ABB RAPID module: Module_Openhole.modx

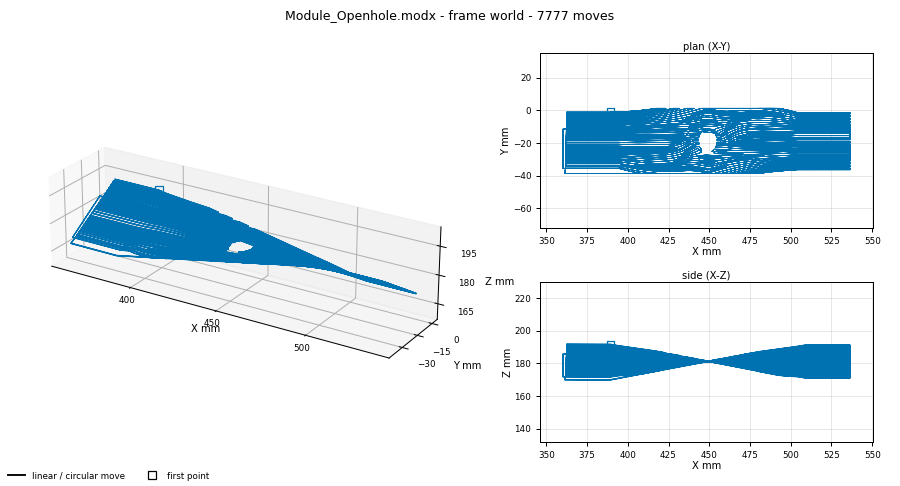
[picture p0: tool path of Module_Openhole.modx in frame world, 7777 of 7777 moves have a stored position in this frame; points joined in program order, loops and branches not executed]
MODULE Module_Openhole

	VAR robtarget Openhole_0 := [[389.38, -1.04, 191.45], [-0.232268, 0.667871, 0.694585, 0.132482], [0,0,0,0], [9E9, 9E9, 9E9, 9E9, 9E9, 9E9]];
	VAR robtarget Openhole_1 := [[394.38, -1.04, 190.58], [-0.220898, 0.671717, 0.697082, 0.118646], [0,0,0,0], [9E9, 9E9, 9E9, 9E9, 9E9, 9E9]];
	VAR robtarget Openhole_2 := [[406.26, -0.14, 188.9], [-0.1941, 0.679945, 0.702469, 0.080853], [0,0,0,0], [9E9, 9E9, 9E9, 9E9, 9E9, 9E9]];
	VAR robtarget Openhole_3 := [[415.11, 0.87, 187.62], [-0.173122, 0.685586, 0.705353, 0.049766], [0,0,0,0], [9E9, 9E9, 9E9, 9E9, 9E9, 9E9]];
	VAR robtarget Openhole_4 := [[417.07, 1.15, 187.33], [-0.16843, 0.686754, 0.705828, 0.042511], [0,0,0,0], [9E9, 9E9, 9E9, 9E9, 9E9, 9E9]];
	VAR robtarget Openhole_5 := [[417.57, 1.3, 187.28], [-0.167467, 0.68699, 0.70595, 0.040437], [0,0,0,0], [9E9, 9E9, 9E9, 9E9, 9E9, 9E9]];
	VAR robtarget Openhole_6 := [[423.41, 1.3, 186.14], [-0.150369, 0.690933, 0.706792, 0.021083], [0,0,0,0], [9E9, 9E9, 9E9, 9E9, 9E9, 9E9]];
	VAR robtarget Openhole_7 := [[422.92, 1.19, 186.21], [-0.151474, 0.690692, 0.70673, 0.023069], [0,0,0,0], [9E9, 9E9, 9E9, 9E9, 9E9, 9E9]];
	VAR robtarget Openhole_8 := [[416.08, 0.05, 187.17], [-0.167887, 0.686887, 0.705392, 0.04921], [0,0,0,0], [9E9, 9E9, 9E9, 9E9, 9E9, 9E9]];
	VAR robtarget Openhole_9 := [[407.72, -0.93, 188.32], [-0.187933, 0.681675, 0.702703, 0.078791], [0,0,0,0], [9E9, 9E9, 9E9, 9E9, 9E9, 9E9]];
	VAR robtarget Openhole_10 := [[395.86, -1.84, 189.92], [-0.215169, 0.673574, 0.697401, 0.116758], [0,0,0,0], [9E9, 9E9, 9E9, 9E9, 9E9, 9E9]];
	VAR robtarget Openhole_11 := [[394.37, -1.93, 190.11], [-0.218405, 0.672532, 0.696636, 0.121237], [0,0,0,0], [9E9, 9E9, 9E9, 9E9, 9E9, 9E9]];
	VAR robtarget Openhole_12 := [[389.38, -1.93, 190.93], [-0.229838, 0.668711, 0.694097, 0.135014], [0,0,0,0], [9E9, 9E9, 9E9, 9E9, 9E9, 9E9]];
	VAR robtarget Openhole_13 := [[362.38, -1.93, 191.02], [-0.183051, 0.683002, 0.683002, 0.183051], [0,0,0,0], [9E9, 9E9, 9E9, 9E9, 9E9, 9E9]];
	VAR robtarget Openhole_14 := [[362.37, -2.82, 190.51], [-0.183051, 0.683002, 0.683002, 0.183051], [0,0,0,0], [9E9, 9E9, 9E9, 9E9, 9E9, 9E9]];
	VAR robtarget Openhole_15 := [[374.37, -2.82, 190.47], [-0.183051, 0.683002, 0.683002, 0.183051], [0,0,0,0], [9E9, 9E9, 9E9, 9E9, 9E9, 9E9]];
	VAR robtarget Openhole_16 := [[389.37, -2.82, 190.42], [-0.227419, 0.669538, 0.693603, 0.137529], [0,0,0,0], [9E9, 9E9, 9E9, 9E9, 9E9, 9E9]];
	VAR robtarget Openhole_17 := [[394.37, -2.82, 189.64], [-0.215931, 0.67333, 0.696182, 0.12382], [0,0,0,0], [9E9, 9E9, 9E9, 9E9, 9E9, 9E9]];
	VAR robtarget Openhole_18 := [[408.22, -1.78, 187.89], [-0.184033, 0.682738, 0.702585, 0.079843], [0,0,0,0], [9E9, 9E9, 9E9, 9E9, 9E9, 9E9]];
	VAR robtarget Openhole_19 := [[416.11, -0.88, 186.87], [-0.164956, 0.687597, 0.705187, 0.052065], [0,0,0,0], [9E9, 9E9, 9E9, 9E9, 9E9, 9E9]];
	VAR robtarget Openhole_20 := [[422.95, 0.24, 185.96], [-0.148411, 0.691357, 0.706629, 0.025979], [0,0,0,0], [9E9, 9E9, 9E9, 9E9, 9E9, 9E9]];
	VAR robtarget Openhole_21 := [[427.32, 1.15, 185.34], [-0.138034, 0.693503, 0.707057, 0.008389], [0,0,0,0], [9E9, 9E9, 9E9, 9E9, 9E9, 9E9]];
	VAR robtarget Openhole_22 := [[427.8, 1.3, 185.28], [-0.137012, 0.693706, 0.707079, 0.006266], [0,0,0,0], [9E9, 9E9, 9E9, 9E9, 9E9, 9E9]];
	VAR robtarget Openhole_23 := [[431.7, 1.3, 184.52], [-0.124848, 0.695998, 0.707072, -0.007002], [0,0,0,0], [9E9, 9E9, 9E9, 9E9, 9E9, 9E9]];
	VAR robtarget Openhole_24 := [[431.22, 1.07, 184.57], [-0.125655, 0.695853, 0.707092, -0.004617], [0,0,0,0], [9E9, 9E9, 9E9, 9E9, 9E9, 9E9]];
	VAR robtarget Openhole_25 := [[423.96, -0.54, 185.58], [-0.142927, 0.692511, 0.706661, 0.025111], [0,0,0,0], [9E9, 9E9, 9E9, 9E9, 9E9, 9E9]];
	VAR robtarget Openhole_26 := [[417.11, -1.69, 186.44], [-0.159586, 0.688863, 0.70524, 0.051343], [0,0,0,0], [9E9, 9E9, 9E9, 9E9, 9E9, 9E9]];
	VAR robtarget Openhole_27 := [[409.22, -2.6, 187.41], [-0.178884, 0.684106, 0.702651, 0.079257], [0,0,0,0], [9E9, 9E9, 9E9, 9E9, 9E9, 9E9]];
	VAR robtarget Openhole_28 := [[394.87, -3.67, 189.12], [-0.212354, 0.674467, 0.695988, 0.124905], [0,0,0,0], [9E9, 9E9, 9E9, 9E9, 9E9, 9E9]];
	VAR robtarget Openhole_29 := [[394.36, -3.7, 189.17], [-0.21345, 0.674121, 0.695717, 0.126406], [0,0,0,0], [9E9, 9E9, 9E9, 9E9, 9E9, 9E9]];
	VAR robtarget Openhole_30 := [[389.37, -3.7, 189.91], [-0.224993, 0.670357, 0.693099, 0.140047], [0,0,0,0], [9E9, 9E9, 9E9, 9E9, 9E9, 9E9]];
	VAR robtarget Openhole_31 := [[362.37, -3.7, 190], [-0.183051, 0.683002, 0.683002, 0.183051], [0,0,0,0], [9E9, 9E9, 9E9, 9E9, 9E9, 9E9]];
	VAR robtarget Openhole_32 := [[362.37, -4.58, 189.49], [-0.183051, 0.683002, 0.683002, 0.183051], [0,0,0,0], [9E9, 9E9, 9E9, 9E9, 9E9, 9E9]];
	VAR robtarget Openhole_33 := [[374.37, -4.58, 189.45], [-0.183051, 0.683002, 0.683002, 0.183051], [0,0,0,0], [9E9, 9E9, 9E9, 9E9, 9E9, 9E9]];
	VAR robtarget Openhole_34 := [[389.37, -4.59, 189.4], [-0.222559, 0.671169, 0.692585, 0.142568], [0,0,0,0], [9E9, 9E9, 9E9, 9E9, 9E9, 9E9]];
	VAR robtarget Openhole_35 := [[394.36, -4.59, 188.71], [-0.210967, 0.674902, 0.69524, 0.129002], [0,0,0,0], [9E9, 9E9, 9E9, 9E9, 9E9, 9E9]];
	VAR robtarget Openhole_36 := [[409.73, -3.48, 186.99], [-0.17483, 0.685153, 0.702519, 0.080416], [0,0,0,0], [9E9, 9E9, 9E9, 9E9, 9E9, 9E9]];
	VAR robtarget Openhole_37 := [[417.63, -2.6, 186.08], [-0.155249, 0.689853, 0.70515, 0.052563], [0,0,0,0], [9E9, 9E9, 9E9, 9E9, 9E9, 9E9]];
	VAR robtarget Openhole_38 := [[424, -1.56, 185.32], [-0.13958, 0.693194, 0.706541, 0.028275], [0,0,0,0], [9E9, 9E9, 9E9, 9E9, 9E9, 9E9]];
	VAR robtarget Openhole_39 := [[430.79, -0.09, 184.44], [-0.12327, 0.696279, 0.707106, 0.000635], [0,0,0,0], [9E9, 9E9, 9E9, 9E9, 9E9, 9E9]];
	VAR robtarget Openhole_40 := [[435.6, 1.08, 183.72], [-0.111729, 0.698224, 0.706834, -0.019623], [0,0,0,0], [9E9, 9E9, 9E9, 9E9, 9E9, 9E9]];
	VAR robtarget Openhole_41 := [[436.08, 1.3, 183.66], [-0.110872, 0.698361, 0.706765, -0.021984], [0,0,0,0], [9E9, 9E9, 9E9, 9E9, 9E9, 9E9]];
	VAR robtarget Openhole_42 := [[440.9, 1.3, 182.71], [-0.095117, 0.70068, 0.706055, -0.038547], [0,0,0,0], [9E9, 9E9, 9E9, 9E9, 9E9, 9E9]];
	VAR robtarget Openhole_43 := [[440.43, 1.14, 182.79], [-0.096181, 0.700535, 0.706169, -0.036397], [0,0,0,0], [9E9, 9E9, 9E9, 9E9, 9E9, 9E9]];
	VAR robtarget Openhole_44 := [[431.79, -1.04, 184.1], [-0.11708, 0.697347, 0.707107, 0.000291], [0,0,0,0], [9E9, 9E9, 9E9, 9E9, 9E9, 9E9]];
	VAR robtarget Openhole_45 := [[425, -2.5, 184.94], [-0.133577, 0.694375, 0.706553, 0.027979], [0,0,0,0], [9E9, 9E9, 9E9, 9E9, 9E9, 9E9]];
	VAR robtarget Openhole_46 := [[418.62, -3.5, 185.66], [-0.149564, 0.691108, 0.705175, 0.052228], [0,0,0,0], [9E9, 9E9, 9E9, 9E9, 9E9, 9E9]];
	VAR robtarget Openhole_47 := [[410.22, -4.4, 186.57], [-0.170741, 0.686183, 0.702365, 0.081753], [0,0,0,0], [9E9, 9E9, 9E9, 9E9, 9E9, 9E9]];
	VAR robtarget Openhole_48 := [[394.37, -5.47, 188.24], [-0.208439, 0.675687, 0.694762, 0.131552], [0,0,0,0], [9E9, 9E9, 9E9, 9E9, 9E9, 9E9]];
	VAR robtarget Openhole_49 := [[389.37, -5.47, 188.89], [-0.220121, 0.671972, 0.692061, 0.14509], [0,0,0,0], [9E9, 9E9, 9E9, 9E9, 9E9, 9E9]];
	VAR robtarget Openhole_50 := [[362.37, -5.47, 188.98], [-0.183051, 0.683002, 0.683002, 0.183051], [0,0,0,0], [9E9, 9E9, 9E9, 9E9, 9E9, 9E9]];
	VAR robtarget Openhole_51 := [[362.37, -6.37, 188.45], [-0.183051, 0.683002, 0.683002, 0.183051], [0,0,0,0], [9E9, 9E9, 9E9, 9E9, 9E9, 9E9]];
	VAR robtarget Openhole_52 := [[374.37, -6.37, 188.42], [-0.183051, 0.683002, 0.683002, 0.183051], [0,0,0,0], [9E9, 9E9, 9E9, 9E9, 9E9, 9E9]];
	VAR robtarget Openhole_53 := [[389.37, -6.37, 188.37], [-0.217615, 0.672788, 0.691514, 0.147675], [0,0,0,0], [9E9, 9E9, 9E9, 9E9, 9E9, 9E9]];
	VAR robtarget Openhole_54 := [[394.35, -6.37, 187.76], [-0.205904, 0.676464, 0.694247, 0.134242], [0,0,0,0], [9E9, 9E9, 9E9, 9E9, 9E9, 9E9]];
	VAR robtarget Openhole_55 := [[411.74, -5.23, 186.06], [-0.163934, 0.687841, 0.702611, 0.079612], [0,0,0,0], [9E9, 9E9, 9E9, 9E9, 9E9, 9E9]];
	VAR robtarget Openhole_56 := [[420.15, -4.36, 185.18], [-0.142311, 0.692638, 0.705338, 0.049989], [0,0,0,0], [9E9, 9E9, 9E9, 9E9, 9E9, 9E9]];
	VAR robtarget Openhole_57 := [[427.03, -3.3, 184.44], [-0.12476, 0.696014, 0.706707, 0.023772], [0,0,0,0], [9E9, 9E9, 9E9, 9E9, 9E9, 9E9]];
	VAR robtarget Openhole_58 := [[432.87, -2.08, 183.75], [-0.110304, 0.69845, 0.707107, 0.000048], [0,0,0,0], [9E9, 9E9, 9E9, 9E9, 9E9, 9E9]];
	VAR robtarget Openhole_59 := [[441.01, 0.05, 182.59], [-0.090709, 0.701264, 0.706248, -0.034832], [0,0,0,0], [9E9, 9E9, 9E9, 9E9, 9E9, 9E9]];
	VAR robtarget Openhole_60 := [[444.81, 1.13, 181.94], [-0.081605, 0.702382, 0.705237, -0.051387], [0,0,0,0], [9E9, 9E9, 9E9, 9E9, 9E9, 9E9]];
	VAR robtarget Openhole_61 := [[445.28, 1.3, 181.86], [-0.080561, 0.702503, 0.705076, -0.053548], [0,0,0,0], [9E9, 9E9, 9E9, 9E9, 9E9, 9E9]];
	VAR robtarget Openhole_62 := [[492.93, 1.3, 172.53], [0.078494, 0.702737, 0.678213, -0.200067], [0,0,0,0], [9E9, 9E9, 9E9, 9E9, 9E9, 9E9]];
	VAR robtarget Openhole_63 := [[497.81, 0.35, 172.02], [0.095716, 0.700599, 0.675215, -0.209963], [0,0,0,0], [9E9, 9E9, 9E9, 9E9, 9E9, 9E9]];
	VAR robtarget Openhole_64 := [[502.17, -0.75, 171.76], [0.111656, 0.698236, 0.672857, -0.217402], [0,0,0,0], [9E9, 9E9, 9E9, 9E9, 9E9, 9E9]];
	VAR robtarget Openhole_65 := [[503.61, -1.18, 171.73], [0.117001, 0.69736, 0.672147, -0.219587], [0,0,0,0], [9E9, 9E9, 9E9, 9E9, 9E9, 9E9]];
	VAR robtarget Openhole_66 := [[504.32, -1.34, 171.7], [0.119471, 0.696941, 0.67175, -0.220799], [0,0,0,0], [9E9, 9E9, 9E9, 9E9, 9E9, 9E9]];
	VAR robtarget Openhole_67 := [[509.31, -1.34, 170.85], [0.183051, 0.683002, 0.683002, -0.183051], [0,0,0,0], [9E9, 9E9, 9E9, 9E9, 9E9, 9E9]];
	VAR robtarget Openhole_68 := [[536.31, -1.34, 170.76], [0.183051, 0.683002, 0.683002, -0.183051], [0,0,0,0], [9E9, 9E9, 9E9, 9E9, 9E9, 9E9]];
	VAR robtarget Openhole_69 := [[536.31, -1.86, 171.07], [0.183051, 0.683002, 0.683002, -0.183051], [0,0,0,0], [9E9, 9E9, 9E9, 9E9, 9E9, 9E9]];
	VAR robtarget Openhole_70 := [[509.31, -1.86, 171.15], [0.183051, 0.683002, 0.683002, -0.183051], [0,0,0,0], [9E9, 9E9, 9E9, 9E9, 9E9, 9E9]];
	VAR robtarget Openhole_71 := [[504.32, -1.86, 171.98], [0.120994, 0.696678, 0.672232, -0.219328], [0,0,0,0], [9E9, 9E9, 9E9, 9E9, 9E9, 9E9]];
	VAR robtarget Openhole_72 := [[503.45, -1.68, 172.02], [0.118004, 0.697191, 0.672724, -0.217813], [0,0,0,0], [9E9, 9E9, 9E9, 9E9, 9E9, 9E9]];
	VAR robtarget Openhole_73 := [[502.98, -1.51, 172.02], [0.116192, 0.697495, 0.672938, -0.217151], [0,0,0,0], [9E9, 9E9, 9E9, 9E9, 9E9, 9E9]];
	VAR robtarget Openhole_74 := [[498.64, -0.34, 172.19], [0.100205, 0.699971, 0.675206, -0.209992], [0,0,0,0], [9E9, 9E9, 9E9, 9E9, 9E9, 9E9]];
	VAR robtarget Openhole_75 := [[493.76, 0.68, 172.63], [0.082548, 0.702272, 0.678031, -0.200682], [0,0,0,0], [9E9, 9E9, 9E9, 9E9, 9E9, 9E9]];
	VAR robtarget Openhole_76 := [[490.83, 1.18, 172.99], [0.071986, 0.703433, 0.679827, -0.194513], [0,0,0,0], [9E9, 9E9, 9E9, 9E9, 9E9, 9E9]];
	VAR robtarget Openhole_77 := [[490.33, 1.3, 173.04], [0.070413, 0.703592, 0.680176, -0.193289], [0,0,0,0], [9E9, 9E9, 9E9, 9E9, 9E9, 9E9]];
	VAR robtarget Openhole_78 := [[480.37, 1.3, 174.99], [0.038399, 0.706063, 0.687393, -0.165806], [0,0,0,0], [9E9, 9E9, 9E9, 9E9, 9E9, 9E9]];
	VAR robtarget Openhole_79 := [[486.26, 0.75, 174.03], [0.058914, 0.704648, 0.683556, -0.180974], [0,0,0,0], [9E9, 9E9, 9E9, 9E9, 9E9, 9E9]];
	VAR robtarget Openhole_80 := [[492.15, -0.08, 173.25], [0.079897, 0.702578, 0.679886, -0.194305], [0,0,0,0], [9E9, 9E9, 9E9, 9E9, 9E9, 9E9]];
	VAR robtarget Openhole_81 := [[497.53, -1.09, 172.74], [0.099178, 0.700117, 0.676708, -0.2051], [0,0,0,0], [9E9, 9E9, 9E9, 9E9, 9E9, 9E9]];
	VAR robtarget Openhole_82 := [[502.86, -2.42, 172.5], [0.118516, 0.697104, 0.673843, -0.214326], [0,0,0,0], [9E9, 9E9, 9E9, 9E9, 9E9, 9E9]];
	VAR robtarget Openhole_83 := [[503.83, -2.67, 172.48], [0.121975, 0.696507, 0.673336, -0.215915], [0,0,0,0], [9E9, 9E9, 9E9, 9E9, 9E9, 9E9]];
	VAR robtarget Openhole_84 := [[504.4, -2.79, 172.45], [0.123921, 0.696164, 0.673011, -0.216923], [0,0,0,0], [9E9, 9E9, 9E9, 9E9, 9E9, 9E9]];
	VAR robtarget Openhole_85 := [[509.32, -2.79, 171.69], [0.183051, 0.683002, 0.683002, -0.183051], [0,0,0,0], [9E9, 9E9, 9E9, 9E9, 9E9, 9E9]];
	VAR robtarget Openhole_86 := [[536.32, -2.79, 171.6], [0.183051, 0.683002, 0.683002, -0.183051], [0,0,0,0], [9E9, 9E9, 9E9, 9E9, 9E9, 9E9]];
	VAR robtarget Openhole_87 := [[536.32, -3.66, 172.1], [0.183051, 0.683002, 0.683002, -0.183051], [0,0,0,0], [9E9, 9E9, 9E9, 9E9, 9E9, 9E9]];
	VAR robtarget Openhole_88 := [[509.32, -3.66, 172.19], [0.183051, 0.683002, 0.683002, -0.183051], [0,0,0,0], [9E9, 9E9, 9E9, 9E9, 9E9, 9E9]];
	VAR robtarget Openhole_89 := [[504.32, -3.66, 172.93], [0.126217, 0.695751, 0.67386, -0.214271], [0,0,0,0], [9E9, 9E9, 9E9, 9E9, 9E9, 9E9]];
	VAR robtarget Openhole_90 := [[503.61, -3.55, 172.97], [0.123897, 0.696168, 0.67429, -0.212914], [0,0,0,0], [9E9, 9E9, 9E9, 9E9, 9E9, 9E9]];
	VAR robtarget Openhole_91 := [[496.78, -2.08, 173.32], [0.099881, 0.700017, 0.678136, -0.200327], [0,0,0,0], [9E9, 9E9, 9E9, 9E9, 9E9, 9E9]];
	VAR robtarget Openhole_92 := [[490.88, -1.1, 173.89], [0.079095, 0.702669, 0.681676, -0.187931], [0,0,0,0], [9E9, 9E9, 9E9, 9E9, 9E9, 9E9]];
	VAR robtarget Openhole_93 := [[484.49, -0.34, 174.74], [0.056636, 0.704835, 0.685689, -0.172716], [0,0,0,0], [9E9, 9E9, 9E9, 9E9, 9E9, 9E9]];
	VAR robtarget Openhole_94 := [[478.08, 0.04, 175.78], [0.034605, 0.70626, 0.6898, -0.155485], [0,0,0,0], [9E9, 9E9, 9E9, 9E9, 9E9, 9E9]];
	VAR robtarget Openhole_95 := [[475.62, 0.08, 176.23], [0.026334, 0.706616, 0.691382, -0.148292], [0,0,0,0], [9E9, 9E9, 9E9, 9E9, 9E9, 9E9]];
	VAR robtarget Openhole_96 := [[475.13, 0.08, 176.32], [0.024701, 0.706675, 0.691699, -0.14681], [0,0,0,0], [9E9, 9E9, 9E9, 9E9, 9E9, 9E9]];
	VAR robtarget Openhole_97 := [[468.75, -0.12, 177.53], [0.003925, 0.707096, 0.695696, -0.126519], [0,0,0,0], [9E9, 9E9, 9E9, 9E9, 9E9, 9E9]];
	VAR robtarget Openhole_98 := [[461.39, -0.49, 178.91], [-0.019926, 0.706826, 0.699751, -0.101727], [0,0,0,0], [9E9, 9E9, 9E9, 9E9, 9E9, 9E9]];
	VAR robtarget Openhole_99 := [[460.9, -0.5, 179], [-0.021584, 0.706777, 0.699986, -0.100097], [0,0,0,0], [9E9, 9E9, 9E9, 9E9, 9E9, 9E9]];
	VAR robtarget Openhole_100 := [[459.91, -0.49, 179.18], [-0.024971, 0.706666, 0.700437, -0.096889], [0,0,0,0], [9E9, 9E9, 9E9, 9E9, 9E9, 9E9]];
	VAR robtarget Openhole_101 := [[457.94, -0.41, 179.52], [-0.031979, 0.706383, 0.701269, -0.090672], [0,0,0,0], [9E9, 9E9, 9E9, 9E9, 9E9, 9E9]];
	VAR robtarget Openhole_102 := [[456.96, -0.33, 179.69], [-0.035593, 0.70621, 0.701651, -0.087669], [0,0,0,0], [9E9, 9E9, 9E9, 9E9, 9E9, 9E9]];
	VAR robtarget Openhole_103 := [[455.49, -0.16, 179.94], [-0.041157, 0.705908, 0.702181, -0.083319], [0,0,0,0], [9E9, 9E9, 9E9, 9E9, 9E9, 9E9]];
	VAR robtarget Openhole_104 := [[454.52, -0.01, 180.11], [-0.044983, 0.705675, 0.702502, -0.080563], [0,0,0,0], [9E9, 9E9, 9E9, 9E9, 9E9, 9E9]];
	VAR robtarget Openhole_105 := [[453.55, 0.19, 180.28], [-0.048932, 0.705412, 0.702794, -0.077981], [0,0,0,0], [9E9, 9E9, 9E9, 9E9, 9E9, 9E9]];
	VAR robtarget Openhole_106 := [[453.08, 0.32, 180.37], [-0.050991, 0.705266, 0.702921, -0.076829], [0,0,0,0], [9E9, 9E9, 9E9, 9E9, 9E9, 9E9]];
	VAR robtarget Openhole_107 := [[451.65, 0.69, 180.62], [-0.057053, 0.704801, 0.703309, -0.07319], [0,0,0,0], [9E9, 9E9, 9E9, 9E9, 9E9, 9E9]];
	VAR robtarget Openhole_108 := [[451.16, 0.77, 180.71], [-0.058985, 0.704642, 0.703448, -0.071844], [0,0,0,0], [9E9, 9E9, 9E9, 9E9, 9E9, 9E9]];
	VAR robtarget Openhole_109 := [[450.68, 0.85, 180.81], [-0.060871, 0.704482, 0.70359, -0.070433], [0,0,0,0], [9E9, 9E9, 9E9, 9E9, 9E9, 9E9]];
	VAR robtarget Openhole_110 := [[450.19, 0.88, 180.9], [-0.062639, 0.704327, 0.703744, -0.06888], [0,0,0,0], [9E9, 9E9, 9E9, 9E9, 9E9, 9E9]];
	VAR robtarget Openhole_111 := [[449.7, 0.9, 180.99], [-0.06438, 0.70417, 0.703897, -0.067293], [0,0,0,0], [9E9, 9E9, 9E9, 9E9, 9E9, 9E9]];
	VAR robtarget Openhole_112 := [[449.21, 0.87, 181.09], [-0.065931, 0.704026, 0.704065, -0.065521], [0,0,0,0], [9E9, 9E9, 9E9, 9E9, 9E9, 9E9]];
	VAR robtarget Openhole_113 := [[448.72, 0.81, 181.18], [-0.067402, 0.703887, 0.704233, -0.063683], [0,0,0,0], [9E9, 9E9, 9E9, 9E9, 9E9, 9E9]];
	VAR robtarget Openhole_114 := [[447.76, 0.61, 181.36], [-0.069985, 0.703635, 0.704579, -0.05974], [0,0,0,0], [9E9, 9E9, 9E9, 9E9, 9E9, 9E9]];
	VAR robtarget Openhole_115 := [[446.8, 0.36, 181.54], [-0.072379, 0.703393, 0.704912, -0.055673], [0,0,0,0], [9E9, 9E9, 9E9, 9E9, 9E9, 9E9]];
	VAR robtarget Openhole_116 := [[438.73, -1.98, 182.8], [-0.091604, 0.701148, 0.706814, -0.02033], [0,0,0,0], [9E9, 9E9, 9E9, 9E9, 9E9, 9E9]];
	VAR robtarget Openhole_117 := [[433.43, -3.29, 183.47], [-0.104537, 0.699337, 0.707104, 0.002109], [0,0,0,0], [9E9, 9E9, 9E9, 9E9, 9E9, 9E9]];
	VAR robtarget Openhole_118 := [[427.08, -4.48, 184.18], [-0.120798, 0.696712, 0.706573, 0.027462], [0,0,0,0], [9E9, 9E9, 9E9, 9E9, 9E9, 9E9]];
	VAR robtarget Openhole_119 := [[419.69, -5.48, 184.93], [-0.140178, 0.693073, 0.704958, 0.055089], [0,0,0,0], [9E9, 9E9, 9E9, 9E9, 9E9, 9E9]];
	VAR robtarget Openhole_120 := [[409.77, -6.33, 185.9], [-0.166065, 0.68733, 0.701464, 0.089152], [0,0,0,0], [9E9, 9E9, 9E9, 9E9, 9E9, 9E9]];
	VAR robtarget Openhole_121 := [[394.35, -7.26, 187.29], [-0.203395, 0.677223, 0.69374, 0.136838], [0,0,0,0], [9E9, 9E9, 9E9, 9E9, 9E9, 9E9]];
	VAR robtarget Openhole_122 := [[389.37, -7.26, 187.86], [-0.215162, 0.673577, 0.69097, 0.150202], [0,0,0,0], [9E9, 9E9, 9E9, 9E9, 9E9, 9E9]];
	VAR robtarget Openhole_123 := [[362.37, -7.26, 187.94], [-0.183051, 0.683002, 0.683002, 0.183051], [0,0,0,0], [9E9, 9E9, 9E9, 9E9, 9E9, 9E9]];
	VAR robtarget Openhole_124 := [[362.37, -8.14, 187.43], [-0.183051, 0.683002, 0.683002, 0.183051], [0,0,0,0], [9E9, 9E9, 9E9, 9E9, 9E9, 9E9]];
	VAR robtarget Openhole_125 := [[374.36, -8.14, 187.4], [-0.183051, 0.683002, 0.683002, 0.183051], [0,0,0,0], [9E9, 9E9, 9E9, 9E9, 9E9, 9E9]];
	VAR robtarget Openhole_126 := [[389.36, -8.14, 187.35], [-0.212703, 0.674357, 0.690416, 0.152729], [0,0,0,0], [9E9, 9E9, 9E9, 9E9, 9E9, 9E9]];
	VAR robtarget Openhole_127 := [[394.35, -8.14, 186.83], [-0.200864, 0.677978, 0.693227, 0.139415], [0,0,0,0], [9E9, 9E9, 9E9, 9E9, 9E9, 9E9]];
	VAR robtarget Openhole_128 := [[411.28, -7.19, 185.4], [-0.159238, 0.688944, 0.701709, 0.087206], [0,0,0,0], [9E9, 9E9, 9E9, 9E9, 9E9, 9E9]];
	VAR robtarget Openhole_129 := [[421.2, -6.39, 184.49], [-0.132741, 0.694536, 0.705109, 0.053119], [0,0,0,0], [9E9, 9E9, 9E9, 9E9, 9E9, 9E9]];
	VAR robtarget Openhole_130 := [[429.59, -5.33, 183.67], [-0.110165, 0.698472, 0.70677, 0.021825], [0,0,0,0], [9E9, 9E9, 9E9, 9E9, 9E9, 9E9]];
	VAR robtarget Openhole_131 := [[435.95, -4.17, 182.98], [-0.09353, 0.700894, 0.707098, -0.003575], [0,0,0,0], [9E9, 9E9, 9E9, 9E9, 9E9, 9E9]];
	VAR robtarget Openhole_132 := [[441.25, -2.83, 182.32], [-0.08048, 0.702512, 0.706625, -0.026102], [0,0,0,0], [9E9, 9E9, 9E9, 9E9, 9E9, 9E9]];
	VAR robtarget Openhole_133 := [[446.48, -1.34, 181.55], [-0.06789, 0.70384, 0.705409, -0.048969], [0,0,0,0], [9E9, 9E9, 9E9, 9E9, 9E9, 9E9]];
	VAR robtarget Openhole_134 := [[447.44, -1.11, 181.39], [-0.065397, 0.704076, 0.705118, -0.052996], [0,0,0,0], [9E9, 9E9, 9E9, 9E9, 9E9, 9E9]];
	VAR robtarget Openhole_135 := [[447.92, -1.01, 181.31], [-0.064108, 0.704195, 0.704966, -0.054981], [0,0,0,0], [9E9, 9E9, 9E9, 9E9, 9E9, 9E9]];
	VAR robtarget Openhole_136 := [[448.41, -0.92, 181.22], [-0.062761, 0.704316, 0.704812, -0.056924], [0,0,0,0], [9E9, 9E9, 9E9, 9E9, 9E9, 9E9]];
	VAR robtarget Openhole_137 := [[448.9, -0.86, 181.14], [-0.061324, 0.704443, 0.704658, -0.058803], [0,0,0,0], [9E9, 9E9, 9E9, 9E9, 9E9, 9E9]];
	VAR robtarget Openhole_138 := [[449.39, -0.83, 181.05], [-0.059734, 0.704579, 0.70451, -0.060549], [0,0,0,0], [9E9, 9E9, 9E9, 9E9, 9E9, 9E9]];
	VAR robtarget Openhole_139 := [[449.88, -0.83, 180.97], [-0.058081, 0.704717, 0.704362, -0.06224], [0,0,0,0], [9E9, 9E9, 9E9, 9E9, 9E9, 9E9]];
	VAR robtarget Openhole_140 := [[450.37, -0.87, 180.88], [-0.056288, 0.704863, 0.704224, -0.063781], [0,0,0,0], [9E9, 9E9, 9E9, 9E9, 9E9, 9E9]];
	VAR robtarget Openhole_141 := [[450.86, -0.92, 180.8], [-0.054451, 0.705007, 0.704088, -0.065265], [0,0,0,0], [9E9, 9E9, 9E9, 9E9, 9E9, 9E9]];
	VAR robtarget Openhole_142 := [[451.35, -1, 180.71], [-0.052532, 0.705153, 0.703959, -0.066646], [0,0,0,0], [9E9, 9E9, 9E9, 9E9, 9E9, 9E9]];
	VAR robtarget Openhole_143 := [[452.32, -1.2, 180.55], [-0.048584, 0.705436, 0.703708, -0.069247], [0,0,0,0], [9E9, 9E9, 9E9, 9E9, 9E9, 9E9]];
	VAR robtarget Openhole_144 := [[452.8, -1.31, 180.47], [-0.046578, 0.705571, 0.703584, -0.070498], [0,0,0,0], [9E9, 9E9, 9E9, 9E9, 9E9, 9E9]];
	VAR robtarget Openhole_145 := [[455.22, -1.78, 180.09], [-0.036759, 0.706151, 0.702891, -0.077096], [0,0,0,0], [9E9, 9E9, 9E9, 9E9, 9E9, 9E9]];
	VAR robtarget Openhole_146 := [[459.15, -2.25, 179.48], [-0.021814, 0.70677, 0.701532, -0.088615], [0,0,0,0], [9E9, 9E9, 9E9, 9E9, 9E9, 9E9]];
	VAR robtarget Openhole_147 := [[459.64, -2.28, 179.4], [-0.020033, 0.706823, 0.701337, -0.090147], [0,0,0,0], [9E9, 9E9, 9E9, 9E9, 9E9, 9E9]];
	VAR robtarget Openhole_148 := [[460.13, -2.3, 179.32], [-0.018281, 0.70687, 0.701135, -0.091707], [0,0,0,0], [9E9, 9E9, 9E9, 9E9, 9E9, 9E9]];
	VAR robtarget Openhole_149 := [[461.12, -2.32, 179.17], [-0.014848, 0.706951, 0.700711, -0.094889], [0,0,0,0], [9E9, 9E9, 9E9, 9E9, 9E9, 9E9]];
	VAR robtarget Openhole_150 := [[466.05, -2.11, 178.34], [0.001206, 0.707106, 0.698251, -0.111559], [0,0,0,0], [9E9, 9E9, 9E9, 9E9, 9E9, 9E9]];
	VAR robtarget Openhole_151 := [[473.41, -1.61, 177.02], [0.024393, 0.706686, 0.693856, -0.136249], [0,0,0,0], [9E9, 9E9, 9E9, 9E9, 9E9, 9E9]];
	VAR robtarget Openhole_152 := [[476.86, -1.55, 176.43], [0.035645, 0.706208, 0.691685, -0.146871], [0,0,0,0], [9E9, 9E9, 9E9, 9E9, 9E9, 9E9]];
	VAR robtarget Openhole_153 := [[477.35, -1.55, 176.35], [0.037279, 0.706123, 0.691373, -0.148336], [0,0,0,0], [9E9, 9E9, 9E9, 9E9, 9E9, 9E9]];
	VAR robtarget Openhole_154 := [[483.28, -1.79, 175.43], [0.057281, 0.704783, 0.687617, -0.164874], [0,0,0,0], [9E9, 9E9, 9E9, 9E9, 9E9, 9E9]];
	VAR robtarget Openhole_155 := [[489.2, -2.35, 174.66], [0.077729, 0.702822, 0.683906, -0.179645], [0,0,0,0], [9E9, 9E9, 9E9, 9E9, 9E9, 9E9]];
	VAR robtarget Openhole_156 := [[496.1, -3.34, 174], [0.101648, 0.699763, 0.67971, -0.194921], [0,0,0,0], [9E9, 9E9, 9E9, 9E9, 9E9, 9E9]];
	VAR robtarget Openhole_157 := [[501.51, -4.28, 173.65], [0.120102, 0.696833, 0.67651, -0.205751], [0,0,0,0], [9E9, 9E9, 9E9, 9E9, 9E9, 9E9]];
	VAR robtarget Openhole_158 := [[503.48, -4.58, 173.53], [0.126548, 0.695691, 0.675311, -0.209654], [0,0,0,0], [9E9, 9E9, 9E9, 9E9, 9E9, 9E9]];
	VAR robtarget Openhole_159 := [[504.32, -4.67, 173.46], [0.129153, 0.695212, 0.674761, -0.211419], [0,0,0,0], [9E9, 9E9, 9E9, 9E9, 9E9, 9E9]];
	VAR robtarget Openhole_160 := [[509.32, -4.67, 172.77], [0.183051, 0.683002, 0.683002, -0.183051], [0,0,0,0], [9E9, 9E9, 9E9, 9E9, 9E9, 9E9]];
	VAR robtarget Openhole_161 := [[536.32, -4.67, 172.69], [0.183051, 0.683002, 0.683002, -0.183051], [0,0,0,0], [9E9, 9E9, 9E9, 9E9, 9E9, 9E9]];
	VAR robtarget Openhole_162 := [[536.32, -5.62, 173.24], [0.183051, 0.683002, 0.683002, -0.183051], [0,0,0,0], [9E9, 9E9, 9E9, 9E9, 9E9, 9E9]];
	VAR robtarget Openhole_163 := [[524.32, -5.62, 173.27], [0.183051, 0.683002, 0.683002, -0.183051], [0,0,0,0], [9E9, 9E9, 9E9, 9E9, 9E9, 9E9]];
	VAR robtarget Openhole_164 := [[509.32, -5.62, 173.32], [0.183051, 0.683002, 0.683002, -0.183051], [0,0,0,0], [9E9, 9E9, 9E9, 9E9, 9E9, 9E9]];
	VAR robtarget Openhole_165 := [[504.32, -5.62, 173.97], [0.1319, 0.694696, 0.675605, -0.208705], [0,0,0,0], [9E9, 9E9, 9E9, 9E9, 9E9, 9E9]];
	VAR robtarget Openhole_166 := [[503.82, -5.61, 174.03], [0.130493, 0.694962, 0.675962, -0.207547], [0,0,0,0], [9E9, 9E9, 9E9, 9E9, 9E9, 9E9]];
	VAR robtarget Openhole_167 := [[498.86, -5.11, 174.43], [0.115013, 0.69769, 0.679175, -0.196776], [0,0,0,0], [9E9, 9E9, 9E9, 9E9, 9E9, 9E9]];
	VAR robtarget Openhole_168 := [[489.97, -3.94, 175.16], [0.084986, 0.701981, 0.684607, -0.176954], [0,0,0,0], [9E9, 9E9, 9E9, 9E9, 9E9, 9E9]];
	VAR robtarget Openhole_169 := [[483.54, -3.35, 175.9], [0.063031, 0.704292, 0.68858, -0.160802], [0,0,0,0], [9E9, 9E9, 9E9, 9E9, 9E9, 9E9]];
	VAR robtarget Openhole_170 := [[478.1, -3.15, 176.67], [0.044814, 0.705685, 0.691968, -0.145535], [0,0,0,0], [9E9, 9E9, 9E9, 9E9, 9E9, 9E9]];
	VAR robtarget Openhole_171 := [[477.6, -3.15, 176.74], [0.043193, 0.705786, 0.692276, -0.144062], [0,0,0,0], [9E9, 9E9, 9E9, 9E9, 9E9, 9E9]];
	VAR robtarget Openhole_172 := [[477.11, -3.15, 176.82], [0.041573, 0.705884, 0.692583, -0.142581], [0,0,0,0], [9E9, 9E9, 9E9, 9E9, 9E9, 9E9]];
	VAR robtarget Openhole_173 := [[471.68, -3.36, 177.69], [0.024304, 0.706689, 0.695916, -0.125306], [0,0,0,0], [9E9, 9E9, 9E9, 9E9, 9E9, 9E9]];
	VAR robtarget Openhole_174 := [[462.34, -4.17, 179.2], [-0.004601, 0.707092, 0.700988, -0.092824], [0,0,0,0], [9E9, 9E9, 9E9, 9E9, 9E9, 9E9]];
	VAR robtarget Openhole_175 := [[459.87, -4.23, 179.56], [-0.012811, 0.706991, 0.702042, -0.084482], [0,0,0,0], [9E9, 9E9, 9E9, 9E9, 9E9, 9E9]];
	VAR robtarget Openhole_176 := [[459.37, -4.22, 179.63], [-0.014523, 0.706958, 0.702234, -0.082867], [0,0,0,0], [9E9, 9E9, 9E9, 9E9, 9E9, 9E9]];
	VAR robtarget Openhole_177 := [[458.38, -4.18, 179.77], [-0.018029, 0.706877, 0.702599, -0.079714], [0,0,0,0], [9E9, 9E9, 9E9, 9E9, 9E9, 9E9]];
	VAR robtarget Openhole_178 := [[457.39, -4.11, 179.91], [-0.021647, 0.706775, 0.702938, -0.076673], [0,0,0,0], [9E9, 9E9, 9E9, 9E9, 9E9, 9E9]];
	VAR robtarget Openhole_179 := [[452.98, -3.48, 180.52], [-0.038778, 0.706043, 0.704209, -0.06395], [0,0,0,0], [9E9, 9E9, 9E9, 9E9, 9E9, 9E9]];
	VAR robtarget Openhole_180 := [[451.03, -3.16, 180.8], [-0.046477, 0.705578, 0.704691, -0.058395], [0,0,0,0], [9E9, 9E9, 9E9, 9E9, 9E9, 9E9]];
	VAR robtarget Openhole_181 := [[450.54, -3.1, 180.88], [-0.048352, 0.705452, 0.70481, -0.056941], [0,0,0,0], [9E9, 9E9, 9E9, 9E9, 9E9, 9E9]];
	VAR robtarget Openhole_182 := [[449.55, -3.01, 181.03], [-0.051994, 0.705193, 0.705049, -0.0539], [0,0,0,0], [9E9, 9E9, 9E9, 9E9, 9E9, 9E9]];
	VAR robtarget Openhole_183 := [[449.06, -3, 181.11], [-0.053711, 0.705064, 0.705173, -0.052264], [0,0,0,0], [9E9, 9E9, 9E9, 9E9, 9E9, 9E9]];
	VAR robtarget Openhole_184 := [[448.57, -3, 181.18], [-0.055374, 0.704935, 0.705296, -0.050571], [0,0,0,0], [9E9, 9E9, 9E9, 9E9, 9E9, 9E9]];
	VAR robtarget Openhole_185 := [[448.07, -3.04, 181.26], [-0.056913, 0.704813, 0.705423, -0.048764], [0,0,0,0], [9E9, 9E9, 9E9, 9E9, 9E9, 9E9]];
	VAR robtarget Openhole_186 := [[447.58, -3.09, 181.33], [-0.05842, 0.704689, 0.705548, -0.04693], [0,0,0,0], [9E9, 9E9, 9E9, 9E9, 9E9, 9E9]];
	VAR robtarget Openhole_187 := [[447.09, -3.15, 181.41], [-0.05986, 0.704568, 0.705671, -0.045042], [0,0,0,0], [9E9, 9E9, 9E9, 9E9, 9E9, 9E9]];
	VAR robtarget Openhole_188 := [[446.11, -3.31, 181.55], [-0.062631, 0.704328, 0.705907, -0.041182], [0,0,0,0], [9E9, 9E9, 9E9, 9E9, 9E9, 9E9]];
	VAR robtarget Openhole_189 := [[437.9, -5.24, 182.58], [-0.083589, 0.702149, 0.707076, -0.006649], [0,0,0,0], [9E9, 9E9, 9E9, 9E9, 9E9, 9E9]];
	VAR robtarget Openhole_190 := [[431.53, -6.32, 183.24], [-0.100765, 0.69989, 0.706862, 0.018588], [0,0,0,0], [9E9, 9E9, 9E9, 9E9, 9E9, 9E9]];
	VAR robtarget Openhole_191 := [[423.12, -7.3, 184.02], [-0.123999, 0.69615, 0.705352, 0.049786], [0,0,0,0], [9E9, 9E9, 9E9, 9E9, 9E9, 9E9]];
	VAR robtarget Openhole_192 := [[413.19, -8.06, 184.88], [-0.151113, 0.690771, 0.702098, 0.084016], [0,0,0,0], [9E9, 9E9, 9E9, 9E9, 9E9, 9E9]];
	VAR robtarget Openhole_193 := [[394.36, -9.02, 186.36], [-0.198303, 0.678731, 0.692709, 0.141966], [0,0,0,0], [9E9, 9E9, 9E9, 9E9, 9E9, 9E9]];
	VAR robtarget Openhole_194 := [[389.36, -9.02, 186.84], [-0.210239, 0.675129, 0.689852, 0.155257], [0,0,0,0], [9E9, 9E9, 9E9, 9E9, 9E9, 9E9]];
	VAR robtarget Openhole_195 := [[362.36, -9.02, 186.92], [-0.183051, 0.683002, 0.683002, 0.183051], [0,0,0,0], [9E9, 9E9, 9E9, 9E9, 9E9, 9E9]];
	VAR robtarget Openhole_196 := [[362.36, -10.02, 186.35], [-0.183051, 0.683002, 0.683002, 0.183051], [0,0,0,0], [9E9, 9E9, 9E9, 9E9, 9E9, 9E9]];
	VAR robtarget Openhole_197 := [[389.36, -10.02, 186.26], [-0.207442, 0.675994, 0.689201, 0.15812], [0,0,0,0], [9E9, 9E9, 9E9, 9E9, 9E9, 9E9]];
	VAR robtarget Openhole_198 := [[394.36, -10.02, 185.83], [-0.195434, 0.679563, 0.692101, 0.1449], [0,0,0,0], [9E9, 9E9, 9E9, 9E9, 9E9, 9E9]];
	VAR robtarget Openhole_199 := [[406.83, -9.43, 184.99], [-0.164737, 0.68765, 0.698856, 0.107708], [0,0,0,0], [9E9, 9E9, 9E9, 9E9, 9E9, 9E9]];
	VAR robtarget Openhole_200 := [[420.76, -8.72, 183.9], [-0.126637, 0.695675, 0.704376, 0.06208], [0,0,0,0], [9E9, 9E9, 9E9, 9E9, 9E9, 9E9]];
	VAR robtarget Openhole_201 := [[431.69, -7.82, 182.97], [-0.095357, 0.700648, 0.706732, 0.023004], [0,0,0,0], [9E9, 9E9, 9E9, 9E9, 9E9, 9E9]];
	VAR robtarget Openhole_202 := [[439.1, -6.9, 182.26], [-0.074168, 0.703206, 0.707088, -0.005195], [0,0,0,0], [9E9, 9E9, 9E9, 9E9, 9E9, 9E9]];
	VAR robtarget Openhole_203 := [[445.46, -5.78, 181.56], [-0.056633, 0.704835, 0.70644, -0.030702], [0,0,0,0], [9E9, 9E9, 9E9, 9E9, 9E9, 9E9]];
	VAR robtarget Openhole_204 := [[446.44, -5.65, 181.44], [-0.053734, 0.705062, 0.706265, -0.034488], [0,0,0,0], [9E9, 9E9, 9E9, 9E9, 9E9, 9E9]];
	VAR robtarget Openhole_205 := [[446.94, -5.6, 181.37], [-0.05223, 0.705175, 0.706173, -0.036337], [0,0,0,0], [9E9, 9E9, 9E9, 9E9, 9E9, 9E9]];
	VAR robtarget Openhole_206 := [[447.43, -5.56, 181.31], [-0.050682, 0.705288, 0.706077, -0.038148], [0,0,0,0], [9E9, 9E9, 9E9, 9E9, 9E9, 9E9]];
	VAR robtarget Openhole_207 := [[447.93, -5.54, 181.25], [-0.049079, 0.705401, 0.70598, -0.039911], [0,0,0,0], [9E9, 9E9, 9E9, 9E9, 9E9, 9E9]];
	VAR robtarget Openhole_208 := [[448.42, -5.54, 181.18], [-0.047412, 0.705516, 0.705881, -0.041612], [0,0,0,0], [9E9, 9E9, 9E9, 9E9, 9E9, 9E9]];
	VAR robtarget Openhole_209 := [[448.92, -5.55, 181.12], [-0.045703, 0.705628, 0.705782, -0.043272], [0,0,0,0], [9E9, 9E9, 9E9, 9E9, 9E9, 9E9]];
	VAR robtarget Openhole_210 := [[450.4, -5.64, 180.92], [-0.040371, 0.705953, 0.705474, -0.048031], [0,0,0,0], [9E9, 9E9, 9E9, 9E9, 9E9, 9E9]];
	VAR robtarget Openhole_211 := [[456.83, -6.26, 180.14], [-0.016424, 0.706916, 0.703866, -0.067618], [0,0,0,0], [9E9, 9E9, 9E9, 9E9, 9E9, 9E9]];
	VAR robtarget Openhole_212 := [[457.32, -6.28, 180.08], [-0.014652, 0.706955, 0.703713, -0.069196], [0,0,0,0], [9E9, 9E9, 9E9, 9E9, 9E9, 9E9]];
	VAR robtarget Openhole_213 := [[457.82, -6.3, 180.02], [-0.012913, 0.706989, 0.703553, -0.070805], [0,0,0,0], [9E9, 9E9, 9E9, 9E9, 9E9, 9E9]];
	VAR robtarget Openhole_214 := [[458.31, -6.3, 179.96], [-0.011217, 0.707018, 0.703385, -0.072456], [0,0,0,0], [9E9, 9E9, 9E9, 9E9, 9E9, 9E9]];
	VAR robtarget Openhole_215 := [[458.81, -6.29, 179.9], [-0.009551, 0.707042, 0.70321, -0.074131], [0,0,0,0], [9E9, 9E9, 9E9, 9E9, 9E9, 9E9]];
	VAR robtarget Openhole_216 := [[459.31, -6.28, 179.84], [-0.007891, 0.707063, 0.703031, -0.075811], [0,0,0,0], [9E9, 9E9, 9E9, 9E9, 9E9, 9E9]];
	VAR robtarget Openhole_217 := [[460.3, -6.24, 179.71], [-0.00466, 0.707091, 0.702653, -0.079238], [0,0,0,0], [9E9, 9E9, 9E9, 9E9, 9E9, 9E9]];
	VAR robtarget Openhole_218 := [[461.29, -6.17, 179.58], [-0.001526, 0.707105, 0.70225, -0.082734], [0,0,0,0], [9E9, 9E9, 9E9, 9E9, 9E9, 9E9]];
	VAR robtarget Openhole_219 := [[463.75, -5.92, 179.24], [0.005986, 0.707081, 0.701141, -0.09166], [0,0,0,0], [9E9, 9E9, 9E9, 9E9, 9E9, 9E9]];
	VAR robtarget Openhole_220 := [[472.09, -4.91, 177.97], [0.030682, 0.706441, 0.696571, -0.121611], [0,0,0,0], [9E9, 9E9, 9E9, 9E9, 9E9, 9E9]];
	VAR robtarget Openhole_221 := [[477.03, -4.63, 177.22], [0.046066, 0.705605, 0.69358, -0.137646], [0,0,0,0], [9E9, 9E9, 9E9, 9E9, 9E9, 9E9]];
	VAR robtarget Openhole_222 := [[478.51, -4.61, 177.01], [0.050849, 0.705276, 0.692669, -0.142163], [0,0,0,0], [9E9, 9E9, 9E9, 9E9, 9E9, 9E9]];
	VAR robtarget Openhole_223 := [[479.01, -4.61, 176.94], [0.052459, 0.705158, 0.692364, -0.143637], [0,0,0,0], [9E9, 9E9, 9E9, 9E9, 9E9, 9E9]];
	VAR robtarget Openhole_224 := [[484.46, -4.79, 176.25], [0.070489, 0.703585, 0.689004, -0.158977], [0,0,0,0], [9E9, 9E9, 9E9, 9E9, 9E9, 9E9]];
	VAR robtarget Openhole_225 := [[491.4, -5.38, 175.54], [0.093788, 0.700859, 0.684732, -0.17647], [0,0,0,0], [9E9, 9E9, 9E9, 9E9, 9E9, 9E9]];
	VAR robtarget Openhole_226 := [[500.82, -6.37, 174.79], [0.124319, 0.696093, 0.678814, -0.19802], [0,0,0,0], [9E9, 9E9, 9E9, 9E9, 9E9, 9E9]];
	VAR robtarget Openhole_227 := [[503.8, -6.51, 174.5], [0.133046, 0.694477, 0.676755, -0.204946], [0,0,0,0], [9E9, 9E9, 9E9, 9E9, 9E9, 9E9]];
	VAR robtarget Openhole_228 := [[504.29, -6.51, 174.44], [0.134414, 0.694214, 0.676391, -0.206143], [0,0,0,0], [9E9, 9E9, 9E9, 9E9, 9E9, 9E9]];
	VAR robtarget Openhole_229 := [[504.32, -6.51, 174.43], [0.1345, 0.694197, 0.67637, -0.206211], [0,0,0,0], [9E9, 9E9, 9E9, 9E9, 9E9, 9E9]];
	VAR robtarget Openhole_230 := [[509.32, -6.51, 173.83], [0.183051, 0.683002, 0.683002, -0.183051], [0,0,0,0], [9E9, 9E9, 9E9, 9E9, 9E9, 9E9]];
	VAR robtarget Openhole_231 := [[536.32, -6.51, 173.75], [0.183051, 0.683002, 0.683002, -0.183051], [0,0,0,0], [9E9, 9E9, 9E9, 9E9, 9E9, 9E9]];
	VAR robtarget Openhole_232 := [[536.32, -7.39, 174.26], [0.183051, 0.683002, 0.683002, -0.183051], [0,0,0,0], [9E9, 9E9, 9E9, 9E9, 9E9, 9E9]];
	VAR robtarget Openhole_233 := [[509.32, -7.39, 174.34], [0.183051, 0.683002, 0.683002, -0.183051], [0,0,0,0], [9E9, 9E9, 9E9, 9E9, 9E9, 9E9]];
	VAR robtarget Openhole_234 := [[504.33, -7.39, 174.9], [0.137077, 0.693693, 0.677133, -0.203694], [0,0,0,0], [9E9, 9E9, 9E9, 9E9, 9E9, 9E9]];
	VAR robtarget Openhole_235 := [[503.78, -7.39, 174.96], [0.135572, 0.693989, 0.677526, -0.202384], [0,0,0,0], [9E9, 9E9, 9E9, 9E9, 9E9, 9E9]];
	VAR robtarget Openhole_236 := [[499.31, -7.22, 175.38], [0.122587, 0.6964, 0.680619, -0.191723], [0,0,0,0], [9E9, 9E9, 9E9, 9E9, 9E9, 9E9]];
	VAR robtarget Openhole_237 := [[487.39, -6.24, 176.38], [0.084188, 0.702077, 0.688112, -0.162795], [0,0,0,0], [9E9, 9E9, 9E9, 9E9, 9E9, 9E9]];
	VAR robtarget Openhole_238 := [[481.43, -5.99, 177.03], [0.064648, 0.704145, 0.691771, -0.146467], [0,0,0,0], [9E9, 9E9, 9E9, 9E9, 9E9, 9E9]];
	VAR robtarget Openhole_239 := [[479.94, -5.98, 177.22], [0.059847, 0.70457, 0.692682, -0.142095], [0,0,0,0], [9E9, 9E9, 9E9, 9E9, 9E9, 9E9]];
	VAR robtarget Openhole_240 := [[479.45, -5.98, 177.28], [0.058261, 0.704702, 0.692986, -0.140609], [0,0,0,0], [9E9, 9E9, 9E9, 9E9, 9E9, 9E9]];
	VAR robtarget Openhole_241 := [[474.99, -6.17, 177.89], [0.044368, 0.705713, 0.695695, -0.126523], [0,0,0,0], [9E9, 9E9, 9E9, 9E9, 9E9, 9E9]];
	VAR robtarget Openhole_242 := [[470.08, -6.73, 178.61], [0.029952, 0.706472, 0.698601, -0.109345], [0,0,0,0], [9E9, 9E9, 9E9, 9E9, 9E9, 9E9]];
	VAR robtarget Openhole_243 := [[463.74, -7.88, 179.52], [0.012476, 0.706997, 0.70196, -0.085155], [0,0,0,0], [9E9, 9E9, 9E9, 9E9, 9E9, 9E9]];
	VAR robtarget Openhole_244 := [[456.91, -9.15, 180.34], [-0.006444, 0.707077, 0.704706, -0.058219], [0,0,0,0], [9E9, 9E9, 9E9, 9E9, 9E9, 9E9]];
	VAR robtarget Openhole_245 := [[453.95, -9.56, 180.64], [-0.01515, 0.706944, 0.70555, -0.04689], [0,0,0,0], [9E9, 9E9, 9E9, 9E9, 9E9, 9E9]];
	VAR robtarget Openhole_246 := [[453.46, -9.61, 180.69], [-0.016637, 0.706911, 0.705672, -0.045022], [0,0,0,0], [9E9, 9E9, 9E9, 9E9, 9E9, 9E9]];
	VAR robtarget Openhole_247 := [[452.96, -9.66, 180.74], [-0.018169, 0.706873, 0.705787, -0.043187], [0,0,0,0], [9E9, 9E9, 9E9, 9E9, 9E9, 9E9]];
	VAR robtarget Openhole_248 := [[451.47, -9.76, 180.87], [-0.022912, 0.706735, 0.706096, -0.037801], [0,0,0,0], [9E9, 9E9, 9E9, 9E9, 9E9, 9E9]];
	VAR robtarget Openhole_249 := [[450.48, -9.77, 180.96], [-0.026255, 0.706619, 0.706271, -0.034372], [0,0,0,0], [9E9, 9E9, 9E9, 9E9, 9E9, 9E9]];
	VAR robtarget Openhole_250 := [[447, -9.62, 181.27], [-0.03858, 0.706054, 0.706732, -0.023019], [0,0,0,0], [9E9, 9E9, 9E9, 9E9, 9E9, 9E9]];
	VAR robtarget Openhole_251 := [[445.01, -9.52, 181.46], [-0.045641, 0.705632, 0.706913, -0.01657], [0,0,0,0], [9E9, 9E9, 9E9, 9E9, 9E9, 9E9]];
	VAR robtarget Openhole_252 := [[443.51, -9.49, 181.6], [-0.050745, 0.705284, 0.707013, -0.011542], [0,0,0,0], [9E9, 9E9, 9E9, 9E9, 9E9, 9E9]];
	VAR robtarget Openhole_253 := [[433.06, -9.93, 182.49], [-0.083926, 0.702109, 0.706649, 0.025431], [0,0,0,0], [9E9, 9E9, 9E9, 9E9, 9E9, 9E9]];
	VAR robtarget Openhole_254 := [[412.13, -10.76, 184.02], [-0.145725, 0.691928, 0.700585, 0.095819], [0,0,0,0], [9E9, 9E9, 9E9, 9E9, 9E9, 9E9]];
	VAR robtarget Openhole_255 := [[397.17, -11.31, 184.94], [-0.184672, 0.682566, 0.6929, 0.141029], [0,0,0,0], [9E9, 9E9, 9E9, 9E9, 9E9, 9E9]];
	VAR robtarget Openhole_256 := [[394.36, -11.45, 185.07], [-0.191326, 0.680731, 0.69121, 0.149091], [0,0,0,0], [9E9, 9E9, 9E9, 9E9, 9E9, 9E9]];
	VAR robtarget Openhole_257 := [[389.36, -11.45, 185.44], [-0.203436, 0.67721, 0.68825, 0.16221], [0,0,0,0], [9E9, 9E9, 9E9, 9E9, 9E9, 9E9]];
	VAR robtarget Openhole_258 := [[360.28, -11.45, 185.53], [-0.183051, 0.683002, 0.683002, 0.183051], [0,0,0,0], [9E9, 9E9, 9E9, 9E9, 9E9, 9E9]];
	VAR robtarget Openhole_259 := [[360.24, -35.51, 171.63], [-0.183051, 0.683002, 0.683002, 0.183051], [0,0,0,0], [9E9, 9E9, 9E9, 9E9, 9E9, 9E9]];
	VAR robtarget Openhole_260 := [[389.32, -35.51, 171.54], [-0.135065, 0.694087, 0.668629, 0.230077], [0,0,0,0], [9E9, 9E9, 9E9, 9E9, 9E9, 9E9]];
	VAR robtarget Openhole_261 := [[394.32, -35.51, 172.34], [-0.121251, 0.696634, 0.67244, 0.218689], [0,0,0,0], [9E9, 9E9, 9E9, 9E9, 9E9, 9E9]];
	VAR robtarget Openhole_262 := [[394.71, -35.54, 172.38], [-0.120058, 0.69684, 0.672716, 0.217839], [0,0,0,0], [9E9, 9E9, 9E9, 9E9, 9E9, 9E9]];
	VAR robtarget Openhole_263 := [[395.19, -35.69, 172.38], [-0.118261, 0.697147, 0.672936, 0.217158], [0,0,0,0], [9E9, 9E9, 9E9, 9E9, 9E9, 9E9]];
	VAR robtarget Openhole_264 := [[399.52, -36.88, 172.5], [-0.102229, 0.699678, 0.675162, 0.210134], [0,0,0,0], [9E9, 9E9, 9E9, 9E9, 9E9, 9E9]];
	VAR robtarget Openhole_265 := [[404.89, -38.02, 172.94], [-0.082728, 0.702251, 0.678231, 0.200007], [0,0,0,0], [9E9, 9E9, 9E9, 9E9, 9E9, 9E9]];
	VAR robtarget Openhole_266 := [[408.32, -38.6, 173.34], [-0.070346, 0.703599, 0.680311, 0.192812], [0,0,0,0], [9E9, 9E9, 9E9, 9E9, 9E9, 9E9]];
	VAR robtarget Openhole_267 := [[408.81, -38.7, 173.39], [-0.068577, 0.703773, 0.680614, 0.191741], [0,0,0,0], [9E9, 9E9, 9E9, 9E9, 9E9, 9E9]];
	VAR robtarget Openhole_268 := [[419.27, -38.7, 175.37], [-0.034862, 0.706247, 0.688133, 0.162705], [0,0,0,0], [9E9, 9E9, 9E9, 9E9, 9E9, 9E9]];
	VAR robtarget Openhole_269 := [[418.78, -38.66, 175.29], [-0.036535, 0.706162, 0.687809, 0.164071], [0,0,0,0], [9E9, 9E9, 9E9, 9E9, 9E9, 9E9]];
	VAR robtarget Openhole_270 := [[412.88, -38.13, 174.36], [-0.057344, 0.704778, 0.684045, 0.179116], [0,0,0,0], [9E9, 9E9, 9E9, 9E9, 9E9, 9E9]];
	VAR robtarget Openhole_271 := [[406.49, -37.23, 173.56], [-0.080198, 0.702544, 0.680106, 0.193534], [0,0,0,0], [9E9, 9E9, 9E9, 9E9, 9E9, 9E9]];
	VAR robtarget Openhole_272 := [[401.11, -36.21, 173.09], [-0.099551, 0.700064, 0.676953, 0.204292], [0,0,0,0], [9E9, 9E9, 9E9, 9E9, 9E9, 9E9]];
	VAR robtarget Openhole_273 := [[395.28, -34.79, 172.86], [-0.120615, 0.696744, 0.673822, 0.214391], [0,0,0,0], [9E9, 9E9, 9E9, 9E9, 9E9, 9E9]];
	VAR robtarget Openhole_274 := [[394.23, -34.53, 172.84], [-0.124345, 0.696088, 0.673269, 0.216121], [0,0,0,0], [9E9, 9E9, 9E9, 9E9, 9E9, 9E9]];
	VAR robtarget Openhole_275 := [[389.32, -34.53, 172.11], [-0.137851, 0.69354, 0.66955, 0.227382], [0,0,0,0], [9E9, 9E9, 9E9, 9E9, 9E9, 9E9]];
	VAR robtarget Openhole_276 := [[362.32, -34.53, 172.19], [-0.183051, 0.683002, 0.683002, 0.183051], [0,0,0,0], [9E9, 9E9, 9E9, 9E9, 9E9, 9E9]];
	VAR robtarget Openhole_277 := [[362.32, -33.65, 172.7], [-0.183051, 0.683002, 0.683002, 0.183051], [0,0,0,0], [9E9, 9E9, 9E9, 9E9, 9E9, 9E9]];
	VAR robtarget Openhole_278 := [[389.32, -33.65, 172.61], [-0.140327, 0.693043, 0.670361, 0.224981], [0,0,0,0], [9E9, 9E9, 9E9, 9E9, 9E9, 9E9]];
	VAR robtarget Openhole_279 := [[394.32, -33.65, 173.32], [-0.126637, 0.695674, 0.674117, 0.213463], [0,0,0,0], [9E9, 9E9, 9E9, 9E9, 9E9, 9E9]];
	VAR robtarget Openhole_280 := [[395, -33.77, 173.35], [-0.124422, 0.696074, 0.674522, 0.212178], [0,0,0,0], [9E9, 9E9, 9E9, 9E9, 9E9, 9E9]];
	VAR robtarget Openhole_281 := [[402.33, -35.28, 173.71], [-0.098691, 0.700186, 0.678664, 0.198533], [0,0,0,0], [9E9, 9E9, 9E9, 9E9, 9E9, 9E9]];
	VAR robtarget Openhole_282 := [[408.72, -36.33, 174.3], [-0.076059, 0.703004, 0.682484, 0.184976], [0,0,0,0], [9E9, 9E9, 9E9, 9E9, 9E9, 9E9]];
	VAR robtarget Openhole_283 := [[414.63, -37, 175.06], [-0.055244, 0.704945, 0.686167, 0.170807], [0,0,0,0], [9E9, 9E9, 9E9, 9E9, 9E9, 9E9]];
	VAR robtarget Openhole_284 := [[420.55, -37.36, 175.98], [-0.034821, 0.706249, 0.68993, 0.154907], [0,0,0,0], [9E9, 9E9, 9E9, 9E9, 9E9, 9E9]];
	VAR robtarget Openhole_285 := [[424, -37.4, 176.58], [-0.023217, 0.706726, 0.692123, 0.144793], [0,0,0,0], [9E9, 9E9, 9E9, 9E9, 9E9, 9E9]];
	VAR robtarget Openhole_286 := [[424.49, -37.4, 176.67], [-0.021585, 0.706777, 0.692436, 0.143293], [0,0,0,0], [9E9, 9E9, 9E9, 9E9, 9E9, 9E9]];
	VAR robtarget Openhole_287 := [[431.37, -37.13, 177.93], [0.000753, 0.707106, 0.69665, 0.121158], [0,0,0,0], [9E9, 9E9, 9E9, 9E9, 9E9, 9E9]];
	VAR robtarget Openhole_288 := [[437.27, -36.86, 178.99], [0.019995, 0.706824, 0.699805, 0.101355], [0,0,0,0], [9E9, 9E9, 9E9, 9E9, 9E9, 9E9]];
	VAR robtarget Openhole_289 := [[437.76, -36.86, 179.07], [0.021674, 0.706775, 0.700037, 0.099744], [0,0,0,0], [9E9, 9E9, 9E9, 9E9, 9E9, 9E9]];
	VAR robtarget Openhole_290 := [[438.25, -36.86, 179.16], [0.023359, 0.706721, 0.700264, 0.098133], [0,0,0,0], [9E9, 9E9, 9E9, 9E9, 9E9, 9E9]];
	VAR robtarget Openhole_291 := [[442.19, -37.1, 179.82], [0.037583, 0.706107, 0.701869, 0.085907], [0,0,0,0], [9E9, 9E9, 9E9, 9E9, 9E9, 9E9]];
	VAR robtarget Openhole_292 := [[443.17, -37.22, 179.98], [0.041331, 0.705898, 0.702212, 0.083052], [0,0,0,0], [9E9, 9E9, 9E9, 9E9, 9E9, 9E9]];
	VAR robtarget Openhole_293 := [[444.14, -37.38, 180.14], [0.045182, 0.705662, 0.702529, 0.080329], [0,0,0,0], [9E9, 9E9, 9E9, 9E9, 9E9, 9E9]];
	VAR robtarget Openhole_294 := [[445.11, -37.59, 180.3], [0.049146, 0.705397, 0.702817, 0.077769], [0,0,0,0], [9E9, 9E9, 9E9, 9E9, 9E9, 9E9]];
	VAR robtarget Openhole_295 := [[446.06, -37.84, 180.47], [0.053219, 0.705101, 0.703076, 0.07539], [0,0,0,0], [9E9, 9E9, 9E9, 9E9, 9E9, 9E9]];
	VAR robtarget Openhole_296 := [[447.02, -38.07, 180.64], [0.057216, 0.704788, 0.70334, 0.072893], [0,0,0,0], [9E9, 9E9, 9E9, 9E9, 9E9, 9E9]];
	VAR robtarget Openhole_297 := [[447.51, -38.14, 180.72], [0.059121, 0.704631, 0.703482, 0.071509], [0,0,0,0], [9E9, 9E9, 9E9, 9E9, 9E9, 9E9]];
	VAR robtarget Openhole_298 := [[447.99, -38.2, 180.81], [0.060976, 0.704473, 0.703628, 0.070058], [0,0,0,0], [9E9, 9E9, 9E9, 9E9, 9E9, 9E9]];
	VAR robtarget Openhole_299 := [[448.49, -38.23, 180.9], [0.062719, 0.70432, 0.703783, 0.068476], [0,0,0,0], [9E9, 9E9, 9E9, 9E9, 9E9, 9E9]];
	VAR robtarget Openhole_300 := [[448.98, -38.23, 180.99], [0.064389, 0.704169, 0.703943, 0.066814], [0,0,0,0], [9E9, 9E9, 9E9, 9E9, 9E9, 9E9]];
	VAR robtarget Openhole_301 := [[449.47, -38.19, 181.08], [0.065901, 0.704029, 0.704112, 0.065008], [0,0,0,0], [9E9, 9E9, 9E9, 9E9, 9E9, 9E9]];
	VAR robtarget Openhole_302 := [[449.95, -38.12, 181.17], [0.06733, 0.703894, 0.704282, 0.063137], [0,0,0,0], [9E9, 9E9, 9E9, 9E9, 9E9, 9E9]];
	VAR robtarget Openhole_303 := [[450.91, -37.89, 181.35], [0.069822, 0.703651, 0.70463, 0.059133], [0,0,0,0], [9E9, 9E9, 9E9, 9E9, 9E9, 9E9]];
	VAR robtarget Openhole_304 := [[459, -35.6, 182.6], [0.089267, 0.701449, 0.706702, 0.023909], [0,0,0,0], [9E9, 9E9, 9E9, 9E9, 9E9, 9E9]];
	VAR robtarget Openhole_305 := [[464.29, -34.25, 183.25], [0.102082, 0.699699, 0.707106, 0.001341], [0,0,0,0], [9E9, 9E9, 9E9, 9E9, 9E9, 9E9]];
	VAR robtarget Openhole_306 := [[471.13, -32.95, 183.98], [0.119555, 0.696926, 0.706625, -0.026086], [0,0,0,0], [9E9, 9E9, 9E9, 9E9, 9E9, 9E9]];
	VAR robtarget Openhole_307 := [[479.02, -31.9, 184.74], [0.140217, 0.693065, 0.704916, -0.055616], [0,0,0,0], [9E9, 9E9, 9E9, 9E9, 9E9, 9E9]];
	VAR robtarget Openhole_308 := [[488.95, -31.06, 185.65], [0.166032, 0.687338, 0.70139, -0.089736], [0,0,0,0], [9E9, 9E9, 9E9, 9E9, 9E9, 9E9]];
	VAR robtarget Openhole_309 := [[504.38, -30.16, 186.96], [0.203244, 0.677268, 0.693614, -0.137475], [0,0,0,0], [9E9, 9E9, 9E9, 9E9, 9E9, 9E9]];
	VAR robtarget Openhole_310 := [[509.37, -30.16, 187.49], [0.183051, 0.683002, 0.683002, -0.183051], [0,0,0,0], [9E9, 9E9, 9E9, 9E9, 9E9, 9E9]];
	VAR robtarget Openhole_311 := [[536.37, -30.16, 187.41], [0.183051, 0.683002, 0.683002, -0.183051], [0,0,0,0], [9E9, 9E9, 9E9, 9E9, 9E9, 9E9]];
	VAR robtarget Openhole_312 := [[536.36, -29.28, 186.9], [0.183051, 0.683002, 0.683002, -0.183051], [0,0,0,0], [9E9, 9E9, 9E9, 9E9, 9E9, 9E9]];
	VAR robtarget Openhole_313 := [[509.36, -29.28, 186.98], [0.183051, 0.683002, 0.683002, -0.183051], [0,0,0,0], [9E9, 9E9, 9E9, 9E9, 9E9, 9E9]];
	VAR robtarget Openhole_314 := [[504.36, -29.28, 186.49], [0.200694, 0.678028, 0.693103, -0.140028], [0,0,0,0], [9E9, 9E9, 9E9, 9E9, 9E9, 9E9]];
	VAR robtarget Openhole_315 := [[485.08, -30.34, 184.95], [0.152962, 0.690364, 0.702572, -0.079956], [0,0,0,0], [9E9, 9E9, 9E9, 9E9, 9E9, 9E9]];
	VAR robtarget Openhole_316 := [[476.14, -31.11, 184.18], [0.12907, 0.695227, 0.705425, -0.048746], [0,0,0,0], [9E9, 9E9, 9E9, 9E9, 9E9, 9E9]];
	VAR robtarget Openhole_317 := [[468.24, -32.14, 183.45], [0.107838, 0.698835, 0.70685, -0.019054], [0,0,0,0], [9E9, 9E9, 9E9, 9E9, 9E9, 9E9]];
	VAR robtarget Openhole_318 := [[461.89, -33.32, 182.79], [0.091228, 0.701197, 0.707077, 0.006455], [0,0,0,0], [9E9, 9E9, 9E9, 9E9, 9E9, 9E9]];
	VAR robtarget Openhole_319 := [[456.11, -34.79, 182.09], [0.077067, 0.702895, 0.706421, 0.031124], [0,0,0,0], [9E9, 9E9, 9E9, 9E9, 9E9, 9E9]];
	VAR robtarget Openhole_320 := [[451.33, -36.06, 181.39], [0.065225, 0.704092, 0.705215, 0.051683], [0,0,0,0], [9E9, 9E9, 9E9, 9E9, 9E9, 9E9]];
	VAR robtarget Openhole_321 := [[450.85, -36.17, 181.31], [0.063938, 0.70421, 0.705067, 0.053671], [0,0,0,0], [9E9, 9E9, 9E9, 9E9, 9E9, 9E9]];
	VAR robtarget Openhole_322 := [[449.87, -36.33, 181.15], [0.061199, 0.704453, 0.704763, 0.05753], [0,0,0,0], [9E9, 9E9, 9E9, 9E9, 9E9, 9E9]];
	VAR robtarget Openhole_323 := [[449.38, -36.38, 181.07], [0.059706, 0.704582, 0.704611, 0.059362], [0,0,0,0], [9E9, 9E9, 9E9, 9E9, 9E9, 9E9]];
	VAR robtarget Openhole_324 := [[448.89, -36.4, 180.99], [0.058085, 0.704717, 0.704463, 0.061084], [0,0,0,0], [9E9, 9E9, 9E9, 9E9, 9E9, 9E9]];
	VAR robtarget Openhole_325 := [[448.4, -36.38, 180.9], [0.056364, 0.704857, 0.704321, 0.062705], [0,0,0,0], [9E9, 9E9, 9E9, 9E9, 9E9, 9E9]];
	VAR robtarget Openhole_326 := [[447.91, -36.33, 180.82], [0.054542, 0.705, 0.704185, 0.064209], [0,0,0,0], [9E9, 9E9, 9E9, 9E9, 9E9, 9E9]];
	VAR robtarget Openhole_327 := [[447.42, -36.26, 180.74], [0.052642, 0.705145, 0.704056, 0.065616], [0,0,0,0], [9E9, 9E9, 9E9, 9E9, 9E9, 9E9]];
	VAR robtarget Openhole_328 := [[446.93, -36.18, 180.66], [0.050711, 0.705286, 0.703927, 0.066979], [0,0,0,0], [9E9, 9E9, 9E9, 9E9, 9E9, 9E9]];
	VAR robtarget Openhole_329 := [[442.57, -35.3, 180], [0.032951, 0.706339, 0.70271, 0.078727], [0,0,0,0], [9E9, 9E9, 9E9, 9E9, 9E9, 9E9]];
	VAR robtarget Openhole_330 := [[440.11, -35, 179.64], [0.023595, 0.706713, 0.701868, 0.085918], [0,0,0,0], [9E9, 9E9, 9E9, 9E9, 9E9, 9E9]];
	VAR robtarget Openhole_331 := [[439.13, -34.94, 179.5], [0.02001, 0.706824, 0.701488, 0.088965], [0,0,0,0], [9E9, 9E9, 9E9, 9E9, 9E9, 9E9]];
	VAR robtarget Openhole_332 := [[437.15, -34.9, 179.2], [0.013125, 0.706985, 0.700653, 0.095317], [0,0,0,0], [9E9, 9E9, 9E9, 9E9, 9E9, 9E9]];
	VAR robtarget Openhole_333 := [[436.65, -34.9, 179.12], [0.011458, 0.707014, 0.700429, 0.09695], [0,0,0,0], [9E9, 9E9, 9E9, 9E9, 9E9, 9E9]];
	VAR robtarget Openhole_334 := [[431.24, -35.21, 178.24], [-0.005937, 0.707082, 0.697626, 0.115406], [0,0,0,0], [9E9, 9E9, 9E9, 9E9, 9E9, 9E9]];
	VAR robtarget Openhole_335 := [[424.35, -35.64, 177.07], [-0.027711, 0.706564, 0.693479, 0.138157], [0,0,0,0], [9E9, 9E9, 9E9, 9E9, 9E9, 9E9]];
	VAR robtarget Openhole_336 := [[421.88, -35.68, 176.66], [-0.035769, 0.706202, 0.691931, 0.145709], [0,0,0,0], [9E9, 9E9, 9E9, 9E9, 9E9, 9E9]];
	VAR robtarget Openhole_337 := [[421.39, -35.68, 176.58], [-0.037405, 0.706117, 0.691621, 0.147175], [0,0,0,0], [9E9, 9E9, 9E9, 9E9, 9E9, 9E9]];
	VAR robtarget Openhole_338 := [[415.95, -35.48, 175.78], [-0.055758, 0.704905, 0.688202, 0.162413], [0,0,0,0], [9E9, 9E9, 9E9, 9E9, 9E9, 9E9]];
	VAR robtarget Openhole_339 := [[410.02, -34.94, 175.04], [-0.076254, 0.702983, 0.684515, 0.177311], [0,0,0,0], [9E9, 9E9, 9E9, 9E9, 9E9, 9E9]];
	VAR robtarget Openhole_340 := [[403.61, -34.06, 174.45], [-0.09857, 0.700203, 0.680636, 0.191662], [0,0,0,0], [9E9, 9E9, 9E9, 9E9, 9E9, 9E9]];
	VAR robtarget Openhole_341 := [[395.25, -32.64, 173.98], [-0.127016, 0.695605, 0.675703, 0.208388], [0,0,0,0], [9E9, 9E9, 9E9, 9E9, 9E9, 9E9]];
	VAR robtarget Openhole_342 := [[394.32, -32.55, 173.9], [-0.129849, 0.695082, 0.675099, 0.210337], [0,0,0,0], [9E9, 9E9, 9E9, 9E9, 9E9, 9E9]];
	VAR robtarget Openhole_343 := [[389.32, -32.55, 173.25], [-0.143464, 0.6924, 0.671376, 0.221934], [0,0,0,0], [9E9, 9E9, 9E9, 9E9, 9E9, 9E9]];
	VAR robtarget Openhole_344 := [[362.32, -32.55, 173.34], [-0.183051, 0.683002, 0.683002, 0.183051], [0,0,0,0], [9E9, 9E9, 9E9, 9E9, 9E9, 9E9]];
	VAR robtarget Openhole_345 := [[362.32, -31.54, 173.92], [-0.183051, 0.683002, 0.683002, 0.183051], [0,0,0,0], [9E9, 9E9, 9E9, 9E9, 9E9, 9E9]];
	VAR robtarget Openhole_346 := [[374.32, -31.54, 173.88], [-0.183051, 0.683002, 0.683002, 0.183051], [0,0,0,0], [9E9, 9E9, 9E9, 9E9, 9E9, 9E9]];
	VAR robtarget Openhole_347 := [[389.32, -31.54, 173.83], [-0.146326, 0.691801, 0.672291, 0.219147], [0,0,0,0], [9E9, 9E9, 9E9, 9E9, 9E9, 9E9]];
	VAR robtarget Openhole_348 := [[394.33, -31.54, 174.44], [-0.13277, 0.69453, 0.675985, 0.20747], [0,0,0,0], [9E9, 9E9, 9E9, 9E9, 9E9, 9E9]];
	VAR robtarget Openhole_349 := [[394.82, -31.57, 174.48], [-0.131308, 0.694808, 0.676325, 0.206362], [0,0,0,0], [9E9, 9E9, 9E9, 9E9, 9E9, 9E9]];
	VAR robtarget Openhole_350 := [[399.78, -32.12, 174.82], [-0.115659, 0.697584, 0.679474, 0.195742], [0,0,0,0], [9E9, 9E9, 9E9, 9E9, 9E9, 9E9]];
	VAR robtarget Openhole_351 := [[407.69, -33.18, 175.39], [-0.088901, 0.701496, 0.684253, 0.178321], [0,0,0,0], [9E9, 9E9, 9E9, 9E9, 9E9, 9E9]];
	VAR robtarget Openhole_352 := [[414.62, -33.85, 176.11], [-0.065169, 0.704097, 0.688491, 0.161183], [0,0,0,0], [9E9, 9E9, 9E9, 9E9, 9E9, 9E9]];
	VAR robtarget Openhole_353 := [[420.07, -34.09, 176.82], [-0.046822, 0.705555, 0.691847, 0.146109], [0,0,0,0], [9E9, 9E9, 9E9, 9E9, 9E9, 9E9]];
	VAR robtarget Openhole_354 := [[421.06, -34.1, 176.96], [-0.043558, 0.705764, 0.692457, 0.143188], [0,0,0,0], [9E9, 9E9, 9E9, 9E9, 9E9, 9E9]];
	VAR robtarget Openhole_355 := [[421.55, -34.1, 177.03], [-0.041935, 0.705862, 0.692762, 0.141706], [0,0,0,0], [9E9, 9E9, 9E9, 9E9, 9E9, 9E9]];
	VAR robtarget Openhole_356 := [[426.98, -33.88, 177.87], [-0.024604, 0.706679, 0.696067, 0.12446], [0,0,0,0], [9E9, 9E9, 9E9, 9E9, 9E9, 9E9]];
	VAR robtarget Openhole_357 := [[436.34, -33.07, 179.3], [0.004346, 0.707093, 0.701098, 0.091983], [0,0,0,0], [9E9, 9E9, 9E9, 9E9, 9E9, 9E9]];
	VAR robtarget Openhole_358 := [[438.32, -33.02, 179.58], [0.010898, 0.707023, 0.701943, 0.085296], [0,0,0,0], [9E9, 9E9, 9E9, 9E9, 9E9, 9E9]];
	VAR robtarget Openhole_359 := [[438.81, -33.02, 179.64], [0.012593, 0.706995, 0.702139, 0.083668], [0,0,0,0], [9E9, 9E9, 9E9, 9E9, 9E9, 9E9]];
	VAR robtarget Openhole_360 := [[439.31, -33.03, 179.71], [0.014313, 0.706962, 0.702329, 0.082061], [0,0,0,0], [9E9, 9E9, 9E9, 9E9, 9E9, 9E9]];
	VAR robtarget Openhole_361 := [[442.77, -33.27, 180.16], [0.02691, 0.706595, 0.7035, 0.071332], [0,0,0,0], [9E9, 9E9, 9E9, 9E9, 9E9, 9E9]];
	VAR robtarget Openhole_362 := [[447.66, -34.06, 180.82], [0.046198, 0.705596, 0.704766, 0.057493], [0,0,0,0], [9E9, 9E9, 9E9, 9E9, 9E9, 9E9]];
	VAR robtarget Openhole_363 := [[448.15, -34.12, 180.89], [0.04807, 0.705471, 0.704883, 0.056034], [0,0,0,0], [9E9, 9E9, 9E9, 9E9, 9E9, 9E9]];
	VAR robtarget Openhole_364 := [[448.65, -34.17, 180.96], [0.049901, 0.705344, 0.705001, 0.054525], [0,0,0,0], [9E9, 9E9, 9E9, 9E9, 9E9, 9E9]];
	VAR robtarget Openhole_365 := [[449.14, -34.2, 181.03], [0.051689, 0.705215, 0.705121, 0.052962], [0,0,0,0], [9E9, 9E9, 9E9, 9E9, 9E9, 9E9]];
	VAR robtarget Openhole_366 := [[449.64, -34.22, 181.1], [0.053409, 0.705087, 0.705241, 0.051328], [0,0,0,0], [9E9, 9E9, 9E9, 9E9, 9E9, 9E9]];
	VAR robtarget Openhole_367 := [[450.13, -34.22, 181.18], [0.055084, 0.704958, 0.705362, 0.049646], [0,0,0,0], [9E9, 9E9, 9E9, 9E9, 9E9, 9E9]];
	VAR robtarget Openhole_368 := [[450.62, -34.2, 181.25], [0.056691, 0.704831, 0.705483, 0.0479], [0,0,0,0], [9E9, 9E9, 9E9, 9E9, 9E9, 9E9]];
	VAR robtarget Openhole_369 := [[451.12, -34.17, 181.32], [0.05825, 0.704703, 0.705602, 0.046108], [0,0,0,0], [9E9, 9E9, 9E9, 9E9, 9E9, 9E9]];
	VAR robtarget Openhole_370 := [[451.61, -34.11, 181.39], [0.059733, 0.704579, 0.705721, 0.044254], [0,0,0,0], [9E9, 9E9, 9E9, 9E9, 9E9, 9E9]];
	VAR robtarget Openhole_371 := [[452.1, -34.05, 181.46], [0.061164, 0.704456, 0.705837, 0.042356], [0,0,0,0], [9E9, 9E9, 9E9, 9E9, 9E9, 9E9]];
	VAR robtarget Openhole_372 := [[452.59, -33.96, 181.53], [0.062536, 0.704336, 0.705951, 0.040416], [0,0,0,0], [9E9, 9E9, 9E9, 9E9, 9E9, 9E9]];
	VAR robtarget Openhole_373 := [[460.82, -32.06, 182.5], [0.083598, 0.702148, 0.707082, 0.005936], [0,0,0,0], [9E9, 9E9, 9E9, 9E9, 9E9, 9E9]];
	VAR robtarget Openhole_374 := [[467.69, -30.95, 183.17], [0.102233, 0.699677, 0.706791, -0.021118], [0,0,0,0], [9E9, 9E9, 9E9, 9E9, 9E9, 9E9]];
	VAR robtarget Openhole_375 := [[476.61, -29.98, 183.94], [0.12687, 0.695632, 0.705046, -0.053948], [0,0,0,0], [9E9, 9E9, 9E9, 9E9, 9E9, 9E9]];
	VAR robtarget Openhole_376 := [[487.55, -29.21, 184.81], [0.15647, 0.689578, 0.701199, -0.091212], [0,0,0,0], [9E9, 9E9, 9E9, 9E9, 9E9, 9E9]];
	VAR robtarget Openhole_377 := [[504.36, -28.38, 186.02], [0.198145, 0.678777, 0.692571, -0.142636], [0,0,0,0], [9E9, 9E9, 9E9, 9E9, 9E9, 9E9]];
	VAR robtarget Openhole_378 := [[509.36, -28.38, 186.47], [0.183051, 0.683002, 0.683002, -0.183051], [0,0,0,0], [9E9, 9E9, 9E9, 9E9, 9E9, 9E9]];
	VAR robtarget Openhole_379 := [[536.36, -28.38, 186.38], [0.183051, 0.683002, 0.683002, -0.183051], [0,0,0,0], [9E9, 9E9, 9E9, 9E9, 9E9, 9E9]];
	VAR robtarget Openhole_380 := [[536.36, -27.26, 185.73], [0.183051, 0.683002, 0.683002, -0.183051], [0,0,0,0], [9E9, 9E9, 9E9, 9E9, 9E9, 9E9]];
	VAR robtarget Openhole_381 := [[509.36, -27.26, 185.82], [0.183051, 0.683002, 0.683002, -0.183051], [0,0,0,0], [9E9, 9E9, 9E9, 9E9, 9E9, 9E9]];
	VAR robtarget Openhole_382 := [[504.36, -27.26, 185.42], [0.194932, 0.679707, 0.691888, -0.145917], [0,0,0,0], [9E9, 9E9, 9E9, 9E9, 9E9, 9E9]];
	VAR robtarget Openhole_383 := [[490.44, -27.87, 184.56], [0.160429, 0.688667, 0.699385, -0.104214], [0,0,0,0], [9E9, 9E9, 9E9, 9E9, 9E9, 9E9]];
	VAR robtarget Openhole_384 := [[476.49, -28.59, 183.56], [0.122048, 0.696494, 0.704715, -0.058112], [0,0,0,0], [9E9, 9E9, 9E9, 9E9, 9E9, 9E9]];
	VAR robtarget Openhole_385 := [[464.07, -29.6, 182.56], [0.086112, 0.701844, 0.70698, -0.013377], [0,0,0,0], [9E9, 9E9, 9E9, 9E9, 9E9, 9E9]];
	VAR robtarget Openhole_386 := [[458.64, -30.3, 182.07], [0.070593, 0.703574, 0.707067, 0.007478], [0,0,0,0], [9E9, 9E9, 9E9, 9E9, 9E9, 9E9]];
	VAR robtarget Openhole_387 := [[453.73, -31.11, 181.57], [0.056891, 0.704814, 0.706592, 0.026972], [0,0,0,0], [9E9, 9E9, 9E9, 9E9, 9E9, 9E9]];
	VAR robtarget Openhole_388 := [[452.74, -31.23, 181.46], [0.053976, 0.705044, 0.706438, 0.030748], [0,0,0,0], [9E9, 9E9, 9E9, 9E9, 9E9, 9E9]];
	VAR robtarget Openhole_389 := [[451.75, -31.32, 181.35], [0.050921, 0.705271, 0.706269, 0.034411], [0,0,0,0], [9E9, 9E9, 9E9, 9E9, 9E9, 9E9]];
	VAR robtarget Openhole_390 := [[450.76, -31.35, 181.23], [0.047689, 0.705497, 0.706089, 0.037916], [0,0,0,0], [9E9, 9E9, 9E9, 9E9, 9E9, 9E9]];
	VAR robtarget Openhole_391 := [[450.27, -31.35, 181.17], [0.046009, 0.705608, 0.705997, 0.039606], [0,0,0,0], [9E9, 9E9, 9E9, 9E9, 9E9, 9E9]];
	VAR robtarget Openhole_392 := [[449.77, -31.34, 181.11], [0.04428, 0.705719, 0.705903, 0.041249], [0,0,0,0], [9E9, 9E9, 9E9, 9E9, 9E9, 9E9]];
	VAR robtarget Openhole_393 := [[449.27, -31.31, 181.05], [0.042523, 0.705827, 0.705807, 0.042861], [0,0,0,0], [9E9, 9E9, 9E9, 9E9, 9E9, 9E9]];
	VAR robtarget Openhole_394 := [[445.32, -30.96, 180.6], [0.027883, 0.706557, 0.704958, 0.05508], [0,0,0,0], [9E9, 9E9, 9E9, 9E9, 9E9, 9E9]];
	VAR robtarget Openhole_395 := [[441.35, -30.75, 180.16], [0.013655, 0.706975, 0.703858, 0.067706], [0,0,0,0], [9E9, 9E9, 9E9, 9E9, 9E9, 9E9]];
	VAR robtarget Openhole_396 := [[440.85, -30.75, 180.1], [0.011961, 0.707006, 0.703696, 0.069364], [0,0,0,0], [9E9, 9E9, 9E9, 9E9, 9E9, 9E9]];
	VAR robtarget Openhole_397 := [[440.35, -30.75, 180.05], [0.010288, 0.707032, 0.703529, 0.071037], [0,0,0,0], [9E9, 9E9, 9E9, 9E9, 9E9, 9E9]];
	VAR robtarget Openhole_398 := [[439.36, -30.78, 179.93], [0.007008, 0.707072, 0.703178, 0.074439], [0,0,0,0], [9E9, 9E9, 9E9, 9E9, 9E9, 9E9]];
	VAR robtarget Openhole_399 := [[438.37, -30.84, 179.81], [0.003826, 0.707096, 0.702801, 0.077914], [0,0,0,0], [9E9, 9E9, 9E9, 9E9, 9E9, 9E9]];
	VAR robtarget Openhole_400 := [[432.46, -31.52, 179.03], [-0.013953, 0.706969, 0.700078, 0.099451], [0,0,0,0], [9E9, 9E9, 9E9, 9E9, 9E9, 9E9]];
	VAR robtarget Openhole_401 := [[426.07, -32.27, 178.1], [-0.03288, 0.706342, 0.696483, 0.122112], [0,0,0,0], [9E9, 9E9, 9E9, 9E9, 9E9, 9E9]];
	VAR robtarget Openhole_402 := [[421.13, -32.53, 177.4], [-0.048367, 0.705451, 0.693508, 0.138007], [0,0,0,0], [9E9, 9E9, 9E9, 9E9, 9E9, 9E9]];
	VAR robtarget Openhole_403 := [[419.64, -32.54, 177.2], [-0.053177, 0.705104, 0.692603, 0.142483], [0,0,0,0], [9E9, 9E9, 9E9, 9E9, 9E9, 9E9]];
	VAR robtarget Openhole_404 := [[419.15, -32.54, 177.14], [-0.054794, 0.704981, 0.6923, 0.143945], [0,0,0,0], [9E9, 9E9, 9E9, 9E9, 9E9, 9E9]];
	VAR robtarget Openhole_405 := [[413.19, -32.29, 176.45], [-0.074612, 0.703159, 0.688673, 0.160406], [0,0,0,0], [9E9, 9E9, 9E9, 9E9, 9E9, 9E9]];
	VAR robtarget Openhole_406 := [[404.76, -31.51, 175.71], [-0.102895, 0.69958, 0.683524, 0.181095], [0,0,0,0], [9E9, 9E9, 9E9, 9E9, 9E9, 9E9]];
	VAR robtarget Openhole_407 := [[397.32, -30.78, 175.18], [-0.126686, 0.695666, 0.678821, 0.197996], [0,0,0,0], [9E9, 9E9, 9E9, 9E9, 9E9, 9E9]];
	VAR robtarget Openhole_408 := [[394.83, -30.66, 174.96], [-0.133955, 0.694302, 0.677113, 0.203759], [0,0,0,0], [9E9, 9E9, 9E9, 9E9, 9E9, 9E9]];
	VAR robtarget Openhole_409 := [[389.32, -30.66, 174.34], [-0.148842, 0.691264, 0.673086, 0.216692], [0,0,0,0], [9E9, 9E9, 9E9, 9E9, 9E9, 9E9]];
	VAR robtarget Openhole_410 := [[362.32, -30.66, 174.43], [-0.183051, 0.683002, 0.683002, 0.183051], [0,0,0,0], [9E9, 9E9, 9E9, 9E9, 9E9, 9E9]];
	VAR robtarget Openhole_411 := [[362.33, -28.99, 175.39], [-0.183051, 0.683002, 0.683002, 0.183051], [0,0,0,0], [9E9, 9E9, 9E9, 9E9, 9E9, 9E9]];
	VAR robtarget Openhole_412 := [[374.33, -28.99, 175.35], [-0.183051, 0.683002, 0.683002, 0.183051], [0,0,0,0], [9E9, 9E9, 9E9, 9E9, 9E9, 9E9]];
	VAR robtarget Openhole_413 := [[389.33, -28.99, 175.31], [-0.153598, 0.690223, 0.674567, 0.212037], [0,0,0,0], [9E9, 9E9, 9E9, 9E9, 9E9, 9E9]];
	VAR robtarget Openhole_414 := [[394.3, -28.99, 175.78], [-0.140299, 0.693049, 0.67816, 0.200246], [0,0,0,0], [9E9, 9E9, 9E9, 9E9, 9E9, 9E9]];
	VAR robtarget Openhole_415 := [[394.82, -28.97, 175.85], [-0.138944, 0.693321, 0.678554, 0.198909], [0,0,0,0], [9E9, 9E9, 9E9, 9E9, 9E9, 9E9]];
	VAR robtarget Openhole_416 := [[396.81, -28.94, 176.05], [-0.133526, 0.694385, 0.679992, 0.193935], [0,0,0,0], [9E9, 9E9, 9E9, 9E9, 9E9, 9E9]];
	VAR robtarget Openhole_417 := [[397.31, -28.94, 176.1], [-0.132135, 0.694651, 0.680344, 0.192696], [0,0,0,0], [9E9, 9E9, 9E9, 9E9, 9E9, 9E9]];
	VAR robtarget Openhole_418 := [[403.29, -29.19, 176.56], [-0.114296, 0.697808, 0.684315, 0.178083], [0,0,0,0], [9E9, 9E9, 9E9, 9E9, 9E9, 9E9]];
	VAR robtarget Openhole_419 := [[414.23, -29.87, 177.4], [-0.078974, 0.702683, 0.691029, 0.14993], [0,0,0,0], [9E9, 9E9, 9E9, 9E9, 9E9, 9E9]];
	VAR robtarget Openhole_420 := [[417.72, -29.94, 177.74], [-0.067712, 0.703857, 0.693111, 0.13999], [0,0,0,0], [9E9, 9E9, 9E9, 9E9, 9E9, 9E9]];
	VAR robtarget Openhole_421 := [[418.21, -29.94, 177.79], [-0.066129, 0.704008, 0.693408, 0.138509], [0,0,0,0], [9E9, 9E9, 9E9, 9E9, 9E9, 9E9]];
	VAR robtarget Openhole_422 := [[423.18, -29.75, 178.36], [-0.050649, 0.70529, 0.696339, 0.122934], [0,0,0,0], [9E9, 9E9, 9E9, 9E9, 9E9, 9E9]];
	VAR robtarget Openhole_423 := [[427.61, -29.25, 178.92], [-0.037686, 0.706102, 0.698891, 0.10748], [0,0,0,0], [9E9, 9E9, 9E9, 9E9, 9E9, 9E9]];
	VAR robtarget Openhole_424 := [[431.99, -28.38, 179.5], [-0.025922, 0.706631, 0.701272, 0.090649], [0,0,0,0], [9E9, 9E9, 9E9, 9E9, 9E9, 9E9]];
	VAR robtarget Openhole_425 := [[436.77, -27.04, 180.09], [-0.014286, 0.706962, 0.703578, 0.070555], [0,0,0,0], [9E9, 9E9, 9E9, 9E9, 9E9, 9E9]];
	VAR robtarget Openhole_426 := [[439.61, -26.14, 180.4], [-0.007686, 0.707065, 0.704719, 0.058065], [0,0,0,0], [9E9, 9E9, 9E9, 9E9, 9E9, 9E9]];
	VAR robtarget Openhole_427 := [[441.02, -25.65, 180.53], [-0.004579, 0.707092, 0.705216, 0.05167], [0,0,0,0], [9E9, 9E9, 9E9, 9E9, 9E9, 9E9]];
	VAR robtarget Openhole_428 := [[441.49, -25.47, 180.57], [-0.003604, 0.707098, 0.705372, 0.049504], [0,0,0,0], [9E9, 9E9, 9E9, 9E9, 9E9, 9E9]];
	VAR robtarget Openhole_429 := [[441.94, -25.27, 180.62], [-0.002734, 0.707101, 0.705524, 0.047292], [0,0,0,0], [9E9, 9E9, 9E9, 9E9, 9E9, 9E9]];
	VAR robtarget Openhole_430 := [[442.83, -24.81, 180.7], [-0.00127, 0.707106, 0.705813, 0.04276], [0,0,0,0], [9E9, 9E9, 9E9, 9E9, 9E9, 9E9]];
	VAR robtarget Openhole_431 := [[443.59, -24.26, 180.77], [-0.000557, 0.707107, 0.706068, 0.038322], [0,0,0,0], [9E9, 9E9, 9E9, 9E9, 9E9, 9E9]];
	VAR robtarget Openhole_432 := [[445.39, -24.26, 180.86], [0.005577, 0.707085, 0.706373, 0.032208], [0,0,0,0], [9E9, 9E9, 9E9, 9E9, 9E9, 9E9]];
	VAR robtarget Openhole_433 := [[443.96, -22.2, 180.9], [-0.006265, 0.707079, 0.706466, 0.030103], [0,0,0,0], [9E9, 9E9, 9E9, 9E9, 9E9, 9E9]];
	VAR robtarget Openhole_434 := [[442.15, -22.2, 180.84], [-0.012387, 0.706998, 0.706179, 0.036212], [0,0,0,0], [9E9, 9E9, 9E9, 9E9, 9E9, 9E9]];
	VAR robtarget Openhole_435 := [[441.31, -22.66, 180.78], [-0.013678, 0.706974, 0.70594, 0.040608], [0,0,0,0], [9E9, 9E9, 9E9, 9E9, 9E9, 9E9]];
	VAR robtarget Openhole_436 := [[440.05, -23.46, 180.66], [-0.015238, 0.706943, 0.705505, 0.04757], [0,0,0,0], [9E9, 9E9, 9E9, 9E9, 9E9, 9E9]];
	VAR robtarget Openhole_437 := [[439.62, -23.72, 180.62], [-0.015821, 0.70693, 0.705346, 0.04987], [0,0,0,0], [9E9, 9E9, 9E9, 9E9, 9E9, 9E9]];
	VAR robtarget Openhole_438 := [[438.31, -24.43, 180.49], [-0.017887, 0.706881, 0.704833, 0.056658], [0,0,0,0], [9E9, 9E9, 9E9, 9E9, 9E9, 9E9]];
	VAR robtarget Openhole_439 := [[435.13, -25.85, 180.13], [-0.023832, 0.706705, 0.703435, 0.071964], [0,0,0,0], [9E9, 9E9, 9E9, 9E9, 9E9, 9E9]];
	VAR robtarget Openhole_440 := [[434.67, -26.03, 180.07], [-0.024783, 0.706672, 0.703214, 0.074093], [0,0,0,0], [9E9, 9E9, 9E9, 9E9, 9E9, 9E9]];
	VAR robtarget Openhole_441 := [[433.73, -26.37, 179.96], [-0.026773, 0.7066, 0.702759, 0.078294], [0,0,0,0], [9E9, 9E9, 9E9, 9E9, 9E9, 9E9]];
	VAR robtarget Openhole_442 := [[432.31, -26.83, 179.78], [-0.030009, 0.70647, 0.702047, 0.084436], [0,0,0,0], [9E9, 9E9, 9E9, 9E9, 9E9, 9E9]];
	VAR robtarget Openhole_443 := [[430.4, -27.35, 179.54], [-0.034677, 0.706256, 0.701049, 0.092361], [0,0,0,0], [9E9, 9E9, 9E9, 9E9, 9E9, 9E9]];
	VAR robtarget Openhole_444 := [[427, -28.06, 179.12], [-0.043621, 0.70576, 0.699187, 0.105533], [0,0,0,0], [9E9, 9E9, 9E9, 9E9, 9E9, 9E9]];
	VAR robtarget Openhole_445 := [[422.56, -28.57, 178.6], [-0.056526, 0.704844, 0.696676, 0.121005], [0,0,0,0], [9E9, 9E9, 9E9, 9E9, 9E9, 9E9]];
	VAR robtarget Openhole_446 := [[417.09, -28.75, 178.04], [-0.073529, 0.703273, 0.693498, 0.13806], [0,0,0,0], [9E9, 9E9, 9E9, 9E9, 9E9, 9E9]];
	VAR robtarget Openhole_447 := [[416.59, -28.75, 178], [-0.07511, 0.703106, 0.693205, 0.139526], [0,0,0,0], [9E9, 9E9, 9E9, 9E9, 9E9, 9E9]];
	VAR robtarget Openhole_448 := [[408.62, -28.45, 177.37], [-0.100727, 0.699896, 0.688444, 0.161386], [0,0,0,0], [9E9, 9E9, 9E9, 9E9, 9E9, 9E9]];
	VAR robtarget Openhole_449 := [[399.66, -28.03, 176.76], [-0.128255, 0.695378, 0.682723, 0.184091], [0,0,0,0], [9E9, 9E9, 9E9, 9E9, 9E9, 9E9]];
	VAR robtarget Openhole_450 := [[398.16, -28.02, 176.63], [-0.132504, 0.694581, 0.681694, 0.187865], [0,0,0,0], [9E9, 9E9, 9E9, 9E9, 9E9, 9E9]];
	VAR robtarget Openhole_451 := [[397.66, -28.02, 176.59], [-0.133885, 0.694316, 0.681343, 0.189133], [0,0,0,0], [9E9, 9E9, 9E9, 9E9, 9E9, 9E9]];
	VAR robtarget Openhole_452 := [[395.18, -28.08, 176.34], [-0.14057, 0.692994, 0.679541, 0.195509], [0,0,0,0], [9E9, 9E9, 9E9, 9E9, 9E9, 9E9]];
	VAR robtarget Openhole_453 := [[394.33, -28.09, 176.26], [-0.142865, 0.692524, 0.678938, 0.197595], [0,0,0,0], [9E9, 9E9, 9E9, 9E9, 9E9, 9E9]];
	VAR robtarget Openhole_454 := [[389.33, -28.09, 175.83], [-0.156171, 0.689645, 0.675356, 0.209511], [0,0,0,0], [9E9, 9E9, 9E9, 9E9, 9E9, 9E9]];
	VAR robtarget Openhole_455 := [[362.33, -28.09, 175.91], [-0.183051, 0.683002, 0.683002, 0.183051], [0,0,0,0], [9E9, 9E9, 9E9, 9E9, 9E9, 9E9]];
	VAR robtarget Openhole_456 := [[362.33, -27.21, 176.42], [-0.183051, 0.683002, 0.683002, 0.183051], [0,0,0,0], [9E9, 9E9, 9E9, 9E9, 9E9, 9E9]];
	VAR robtarget Openhole_457 := [[374.33, -27.21, 176.38], [-0.183051, 0.683002, 0.683002, 0.183051], [0,0,0,0], [9E9, 9E9, 9E9, 9E9, 9E9, 9E9]];
	VAR robtarget Openhole_458 := [[389.33, -27.21, 176.34], [-0.15869, 0.68907, 0.676119, 0.207034], [0,0,0,0], [9E9, 9E9, 9E9, 9E9, 9E9, 9E9]];
	VAR robtarget Openhole_459 := [[394.26, -27.21, 176.73], [-0.145654, 0.691943, 0.679619, 0.195239], [0,0,0,0], [9E9, 9E9, 9E9, 9E9, 9E9, 9E9]];
	VAR robtarget Openhole_460 := [[399.8, -27.04, 177.24], [-0.130818, 0.6949, 0.683607, 0.180779], [0,0,0,0], [9E9, 9E9, 9E9, 9E9, 9E9, 9E9]];
	VAR robtarget Openhole_461 := [[400.3, -27.04, 177.28], [-0.129407, 0.695165, 0.683947, 0.179488], [0,0,0,0], [9E9, 9E9, 9E9, 9E9, 9E9, 9E9]];
	VAR robtarget Openhole_462 := [[416.26, -27.54, 178.35], [-0.080038, 0.702562, 0.693768, 0.136695], [0,0,0,0], [9E9, 9E9, 9E9, 9E9, 9E9, 9E9]];
	VAR robtarget Openhole_463 := [[416.76, -27.54, 178.39], [-0.07846, 0.70274, 0.694056, 0.135227], [0,0,0,0], [9E9, 9E9, 9E9, 9E9, 9E9, 9E9]];
	VAR robtarget Openhole_464 := [[417.25, -27.54, 178.43], [-0.076892, 0.702914, 0.694344, 0.133741], [0,0,0,0], [9E9, 9E9, 9E9, 9E9, 9E9, 9E9]];
	VAR robtarget Openhole_465 := [[422.73, -27.32, 178.94], [-0.060035, 0.704554, 0.697448, 0.116475], [0,0,0,0], [9E9, 9E9, 9E9, 9E9, 9E9, 9E9]];
	VAR robtarget Openhole_466 := [[426.67, -26.85, 179.36], [-0.048682, 0.705429, 0.699624, 0.102595], [0,0,0,0], [9E9, 9E9, 9E9, 9E9, 9E9, 9E9]];
	VAR robtarget Openhole_467 := [[430.07, -26.09, 179.75], [-0.039951, 0.705977, 0.701448, 0.089277], [0,0,0,0], [9E9, 9E9, 9E9, 9E9, 9E9, 9E9]];
	VAR robtarget Openhole_468 := [[432.91, -25.19, 180.09], [-0.033494, 0.706313, 0.702896, 0.077053], [0,0,0,0], [9E9, 9E9, 9E9, 9E9, 9E9, 9E9]];
	VAR robtarget Openhole_469 := [[433.37, -25.01, 180.14], [-0.03254, 0.706358, 0.703125, 0.074938], [0,0,0,0], [9E9, 9E9, 9E9, 9E9, 9E9, 9E9]];
	VAR robtarget Openhole_470 := [[433.83, -24.82, 180.2], [-0.031632, 0.706399, 0.703349, 0.072799], [0,0,0,0], [9E9, 9E9, 9E9, 9E9, 9E9, 9E9]];
	VAR robtarget Openhole_471 := [[434.29, -24.62, 180.25], [-0.030763, 0.706437, 0.70357, 0.070639], [0,0,0,0], [9E9, 9E9, 9E9, 9E9, 9E9, 9E9]];
	VAR robtarget Openhole_472 := [[435.19, -24.2, 180.36], [-0.029143, 0.706506, 0.703995, 0.06626], [0,0,0,0], [9E9, 9E9, 9E9, 9E9, 9E9, 9E9]];
	VAR robtarget Openhole_473 := [[436.52, -23.52, 180.51], [-0.02696, 0.706593, 0.704593, 0.059574], [0,0,0,0], [9E9, 9E9, 9E9, 9E9, 9E9, 9E9]];
	VAR robtarget Openhole_474 := [[438.24, -22.52, 180.69], [-0.024535, 0.706681, 0.705304, 0.050458], [0,0,0,0], [9E9, 9E9, 9E9, 9E9, 9E9, 9E9]];
	VAR robtarget Openhole_475 := [[440.79, -20.96, 180.9], [-0.02119, 0.706789, 0.706159, 0.036601], [0,0,0,0], [9E9, 9E9, 9E9, 9E9, 9E9, 9E9]];
	VAR robtarget Openhole_476 := [[441.58, -20.63, 180.94], [-0.019628, 0.706834, 0.706345, 0.032812], [0,0,0,0], [9E9, 9E9, 9E9, 9E9, 9E9, 9E9]];
	VAR robtarget Openhole_477 := [[443.72, -20.63, 180.97], [-0.012375, 0.706998, 0.706645, 0.02556], [0,0,0,0], [9E9, 9E9, 9E9, 9E9, 9E9, 9E9]];
	VAR robtarget Openhole_478 := [[443.53, -19.52, 181.03], [-0.0168, 0.706907, 0.706751, 0.022442], [0,0,0,0], [9E9, 9E9, 9E9, 9E9, 9E9, 9E9]];
	VAR robtarget Openhole_479 := [[441.39, -19.52, 181.02], [-0.024045, 0.706698, 0.706483, 0.029698], [0,0,0,0], [9E9, 9E9, 9E9, 9E9, 9E9, 9E9]];
	VAR robtarget Openhole_480 := [[440.77, -19.7, 181.01], [-0.025533, 0.706646, 0.706366, 0.032366], [0,0,0,0], [9E9, 9E9, 9E9, 9E9, 9E9, 9E9]];
	VAR robtarget Openhole_481 := [[440.31, -19.89, 180.99], [-0.026411, 0.706613, 0.70626, 0.034586], [0,0,0,0], [9E9, 9E9, 9E9, 9E9, 9E9, 9E9]];
	VAR robtarget Openhole_482 := [[439.86, -20.1, 180.96], [-0.027231, 0.706582, 0.706147, 0.036826], [0,0,0,0], [9E9, 9E9, 9E9, 9E9, 9E9, 9E9]];
	VAR robtarget Openhole_483 := [[439.41, -20.32, 180.94], [-0.028004, 0.706552, 0.706026, 0.039079], [0,0,0,0], [9E9, 9E9, 9E9, 9E9, 9E9, 9E9]];
	VAR robtarget Openhole_484 := [[438.97, -20.55, 180.91], [-0.028703, 0.706524, 0.705897, 0.041353], [0,0,0,0], [9E9, 9E9, 9E9, 9E9, 9E9, 9E9]];
	VAR robtarget Openhole_485 := [[438.54, -20.81, 180.88], [-0.029274, 0.706501, 0.705758, 0.04366], [0,0,0,0], [9E9, 9E9, 9E9, 9E9, 9E9, 9E9]];
	VAR robtarget Openhole_486 := [[436.45, -22.16, 180.67], [-0.031755, 0.706393, 0.704947, 0.055221], [0,0,0,0], [9E9, 9E9, 9E9, 9E9, 9E9, 9E9]];
	VAR robtarget Openhole_487 := [[436.02, -22.42, 180.63], [-0.032352, 0.706366, 0.704765, 0.057498], [0,0,0,0], [9E9, 9E9, 9E9, 9E9, 9E9, 9E9]];
	VAR robtarget Openhole_488 := [[435.15, -22.9, 180.53], [-0.033663, 0.706305, 0.704383, 0.062006], [0,0,0,0], [9E9, 9E9, 9E9, 9E9, 9E9, 9E9]];
	VAR robtarget Openhole_489 := [[434.26, -23.35, 180.43], [-0.035128, 0.706234, 0.703978, 0.066449], [0,0,0,0], [9E9, 9E9, 9E9, 9E9, 9E9, 9E9]];
	VAR robtarget Openhole_490 := [[433.36, -23.77, 180.33], [-0.036731, 0.706152, 0.703551, 0.070826], [0,0,0,0], [9E9, 9E9, 9E9, 9E9, 9E9, 9E9]];
	VAR robtarget Openhole_491 := [[432.44, -24.15, 180.23], [-0.038517, 0.706057, 0.703106, 0.075113], [0,0,0,0], [9E9, 9E9, 9E9, 9E9, 9E9, 9E9]];
	VAR robtarget Openhole_492 := [[431.98, -24.33, 180.18], [-0.039474, 0.706004, 0.702877, 0.077222], [0,0,0,0], [9E9, 9E9, 9E9, 9E9, 9E9, 9E9]];
	VAR robtarget Openhole_493 := [[431.04, -24.65, 180.07], [-0.041547, 0.705885, 0.702412, 0.08135], [0,0,0,0], [9E9, 9E9, 9E9, 9E9, 9E9, 9E9]];
	VAR robtarget Openhole_494 := [[428.64, -25.31, 179.81], [-0.047268, 0.705525, 0.701189, 0.091287], [0,0,0,0], [9E9, 9E9, 9E9, 9E9, 9E9, 9E9]];
	VAR robtarget Openhole_495 := [[426.69, -25.72, 179.6], [-0.05235, 0.705166, 0.700166, 0.098828], [0,0,0,0], [9E9, 9E9, 9E9, 9E9, 9E9, 9E9]];
	VAR robtarget Openhole_496 := [[422.74, -26.21, 179.22], [-0.063627, 0.704238, 0.69805, 0.112808], [0,0,0,0], [9E9, 9E9, 9E9, 9E9, 9E9, 9E9]];
	VAR robtarget Openhole_497 := [[417.76, -26.42, 178.82], [-0.078878, 0.702694, 0.695305, 0.128653], [0,0,0,0], [9E9, 9E9, 9E9, 9E9, 9E9, 9E9]];
	VAR robtarget Openhole_498 := [[416.77, -26.42, 178.74], [-0.082009, 0.702335, 0.694744, 0.131646], [0,0,0,0], [9E9, 9E9, 9E9, 9E9, 9E9, 9E9]];
	VAR robtarget Openhole_499 := [[416.27, -26.42, 178.71], [-0.083581, 0.70215, 0.694462, 0.133124], [0,0,0,0], [9E9, 9E9, 9E9, 9E9, 9E9, 9E9]];
	VAR robtarget Openhole_500 := [[401.3, -26.08, 177.8], [-0.129473, 0.695152, 0.685358, 0.174023], [0,0,0,0], [9E9, 9E9, 9E9, 9E9, 9E9, 9E9]];
	VAR robtarget Openhole_501 := [[400.8, -26.08, 177.77], [-0.130883, 0.694888, 0.685023, 0.175339], [0,0,0,0], [9E9, 9E9, 9E9, 9E9, 9E9, 9E9]];
	VAR robtarget Openhole_502 := [[395.33, -26.26, 177.3], [-0.145541, 0.691967, 0.681142, 0.189857], [0,0,0,0], [9E9, 9E9, 9E9, 9E9, 9E9, 9E9]];
	VAR robtarget Openhole_503 := [[394.83, -26.28, 177.25], [-0.146803, 0.6917, 0.680774, 0.191173], [0,0,0,0], [9E9, 9E9, 9E9, 9E9, 9E9, 9E9]];
	VAR robtarget Openhole_504 := [[394.33, -26.32, 177.2], [-0.148041, 0.691436, 0.680392, 0.192527], [0,0,0,0], [9E9, 9E9, 9E9, 9E9, 9E9, 9E9]];
	VAR robtarget Openhole_505 := [[394.33, -26.32, 177.2], [-0.148023, 0.69144, 0.680396, 0.192512], [0,0,0,0], [9E9, 9E9, 9E9, 9E9, 9E9, 9E9]];
	VAR robtarget Openhole_506 := [[389.33, -26.32, 176.85], [-0.161205, 0.688486, 0.676873, 0.204556], [0,0,0,0], [9E9, 9E9, 9E9, 9E9, 9E9, 9E9]];
	VAR robtarget Openhole_507 := [[362.33, -26.32, 176.93], [-0.183051, 0.683002, 0.683002, 0.183051], [0,0,0,0], [9E9, 9E9, 9E9, 9E9, 9E9, 9E9]];
	VAR robtarget Openhole_508 := [[362.34, -24.22, 178.15], [-0.183051, 0.683002, 0.683002, 0.183051], [0,0,0,0], [9E9, 9E9, 9E9, 9E9, 9E9, 9E9]];
	VAR robtarget Openhole_509 := [[389.34, -24.22, 178.06], [-0.167213, 0.687051, 0.678639, 0.198617], [0,0,0,0], [9E9, 9E9, 9E9, 9E9, 9E9, 9E9]];
	VAR robtarget Openhole_510 := [[394.34, -24.22, 178.31], [-0.154181, 0.690093, 0.682091, 0.18642], [0,0,0,0], [9E9, 9E9, 9E9, 9E9, 9E9, 9E9]];
	VAR robtarget Openhole_511 := [[395.3, -24.2, 178.37], [-0.151654, 0.690653, 0.682766, 0.183929], [0,0,0,0], [9E9, 9E9, 9E9, 9E9, 9E9, 9E9]];
	VAR robtarget Openhole_512 := [[401.29, -23.97, 178.77], [-0.135881, 0.693928, 0.686917, 0.167767], [0,0,0,0], [9E9, 9E9, 9E9, 9E9, 9E9, 9E9]];
	VAR robtarget Openhole_513 := [[403.28, -23.96, 178.87], [-0.130263, 0.695005, 0.688215, 0.162359], [0,0,0,0], [9E9, 9E9, 9E9, 9E9, 9E9, 9E9]];
	VAR robtarget Openhole_514 := [[403.78, -23.96, 178.9], [-0.128833, 0.695271, 0.688533, 0.161004], [0,0,0,0], [9E9, 9E9, 9E9, 9E9, 9E9, 9E9]];
	VAR robtarget Openhole_515 := [[416.77, -24.13, 179.46], [-0.089339, 0.70144, 0.696085, 0.12436], [0,0,0,0], [9E9, 9E9, 9E9, 9E9, 9E9, 9E9]];
	VAR robtarget Openhole_516 := [[417.27, -24.13, 179.49], [-0.087782, 0.701637, 0.696353, 0.122853], [0,0,0,0], [9E9, 9E9, 9E9, 9E9, 9E9, 9E9]];
	VAR robtarget Openhole_517 := [[422.76, -23.95, 179.8], [-0.070952, 0.703538, 0.699201, 0.10544], [0,0,0,0], [9E9, 9E9, 9E9, 9E9, 9E9, 9E9]];
	VAR robtarget Openhole_518 := [[426.72, -23.49, 180.09], [-0.059614, 0.704589, 0.70117, 0.091434], [0,0,0,0], [9E9, 9E9, 9E9, 9E9, 9E9, 9E9]];
	VAR robtarget Openhole_519 := [[427.7, -23.31, 180.17], [-0.057001, 0.704806, 0.701647, 0.087703], [0,0,0,0], [9E9, 9E9, 9E9, 9E9, 9E9, 9E9]];
	VAR robtarget Openhole_520 := [[428.19, -23.21, 180.21], [-0.055737, 0.704907, 0.701882, 0.085798], [0,0,0,0], [9E9, 9E9, 9E9, 9E9, 9E9, 9E9]];
	VAR robtarget Openhole_521 := [[430.12, -22.73, 180.38], [-0.050959, 0.705268, 0.702797, 0.077955], [0,0,0,0], [9E9, 9E9, 9E9, 9E9, 9E9, 9E9]];
	VAR robtarget Openhole_522 := [[430.6, -22.59, 180.42], [-0.049836, 0.705348, 0.703017, 0.075938], [0,0,0,0], [9E9, 9E9, 9E9, 9E9, 9E9, 9E9]];
	VAR robtarget Openhole_523 := [[432.02, -22.13, 180.54], [-0.046655, 0.705566, 0.703657, 0.069758], [0,0,0,0], [9E9, 9E9, 9E9, 9E9, 9E9, 9E9]];
	VAR robtarget Openhole_524 := [[432.49, -21.97, 180.58], [-0.045648, 0.705632, 0.703862, 0.067661], [0,0,0,0], [9E9, 9E9, 9E9, 9E9, 9E9, 9E9]];
	VAR robtarget Openhole_525 := [[433.88, -21.41, 180.71], [-0.042886, 0.705805, 0.704451, 0.061226], [0,0,0,0], [9E9, 9E9, 9E9, 9E9, 9E9, 9E9]];
	VAR robtarget Openhole_526 := [[434.78, -20.99, 180.79], [-0.041291, 0.7059, 0.70482, 0.056817], [0,0,0,0], [9E9, 9E9, 9E9, 9E9, 9E9, 9E9]];
	VAR robtarget Openhole_527 := [[435.23, -20.76, 180.83], [-0.040575, 0.705942, 0.704997, 0.054577], [0,0,0,0], [9E9, 9E9, 9E9, 9E9, 9E9, 9E9]];
	VAR robtarget Openhole_528 := [[436.1, -20.28, 180.9], [-0.039281, 0.706015, 0.705334, 0.050045], [0,0,0,0], [9E9, 9E9, 9E9, 9E9, 9E9, 9E9]];
	VAR robtarget Openhole_529 := [[436.54, -20.05, 180.94], [-0.038588, 0.706053, 0.70549, 0.047786], [0,0,0,0], [9E9, 9E9, 9E9, 9E9, 9E9, 9E9]];
	VAR robtarget Openhole_530 := [[436.99, -19.83, 180.97], [-0.037802, 0.706096, 0.705638, 0.045554], [0,0,0,0], [9E9, 9E9, 9E9, 9E9, 9E9, 9E9]];
	VAR robtarget Openhole_531 := [[437.9, -19.41, 181.02], [-0.036164, 0.706181, 0.705911, 0.041103], [0,0,0,0], [9E9, 9E9, 9E9, 9E9, 9E9, 9E9]];
	VAR robtarget Openhole_532 := [[438.36, -19.23, 181.04], [-0.035217, 0.706229, 0.706035, 0.038923], [0,0,0,0], [9E9, 9E9, 9E9, 9E9, 9E9, 9E9]];
	VAR robtarget Openhole_533 := [[438.83, -19.07, 181.06], [-0.034173, 0.706281, 0.706149, 0.036785], [0,0,0,0], [9E9, 9E9, 9E9, 9E9, 9E9, 9E9]];
	VAR robtarget Openhole_534 := [[439.31, -18.93, 181.07], [-0.033055, 0.706334, 0.706256, 0.034683], [0,0,0,0], [9E9, 9E9, 9E9, 9E9, 9E9, 9E9]];
	VAR robtarget Openhole_535 := [[440.28, -18.68, 181.09], [-0.030631, 0.706443, 0.706446, 0.030573], [0,0,0,0], [9E9, 9E9, 9E9, 9E9, 9E9, 9E9]];
	VAR robtarget Openhole_536 := [[440.77, -18.58, 181.1], [-0.0293, 0.706499, 0.706529, 0.02859], [0,0,0,0], [9E9, 9E9, 9E9, 9E9, 9E9, 9E9]];
	VAR robtarget Openhole_537 := [[441.27, -18.53, 181.1], [-0.027786, 0.706561, 0.706601, 0.026741], [0,0,0,0], [9E9, 9E9, 9E9, 9E9, 9E9, 9E9]];
	VAR robtarget Openhole_538 := [[441.35, -18.53, 181.1], [-0.027522, 0.706571, 0.706611, 0.026486], [0,0,0,0], [9E9, 9E9, 9E9, 9E9, 9E9, 9E9]];
	VAR robtarget Openhole_539 := [[443.12, -18.53, 181.09], [-0.021525, 0.706779, 0.70681, 0.020471], [0,0,0,0], [9E9, 9E9, 9E9, 9E9, 9E9, 9E9]];
	VAR robtarget Openhole_540 := [[443.2, -17.55, 181.15], [-0.024585, 0.706679, 0.706906, 0.016845], [0,0,0,0], [9E9, 9E9, 9E9, 9E9, 9E9, 9E9]];
	VAR robtarget Openhole_541 := [[441.43, -17.55, 181.17], [-0.030578, 0.706445, 0.706737, 0.022866], [0,0,0,0], [9E9, 9E9, 9E9, 9E9, 9E9, 9E9]];
	VAR robtarget Openhole_542 := [[441.36, -17.54, 181.18], [-0.030825, 0.706435, 0.706731, 0.023051], [0,0,0,0], [9E9, 9E9, 9E9, 9E9, 9E9, 9E9]];
	VAR robtarget Openhole_543 := [[440.87, -17.63, 181.18], [-0.032199, 0.706373, 0.706664, 0.025008], [0,0,0,0], [9E9, 9E9, 9E9, 9E9, 9E9, 9E9]];
	VAR robtarget Openhole_544 := [[436.92, -18.24, 181.16], [-0.043395, 0.705774, 0.705951, 0.040414], [0,0,0,0], [9E9, 9E9, 9E9, 9E9, 9E9, 9E9]];
	VAR robtarget Openhole_545 := [[436.43, -18.34, 181.15], [-0.044705, 0.705692, 0.705835, 0.042387], [0,0,0,0], [9E9, 9E9, 9E9, 9E9, 9E9, 9E9]];
	VAR robtarget Openhole_546 := [[435.94, -18.42, 181.14], [-0.046086, 0.705603, 0.705717, 0.044307], [0,0,0,0], [9E9, 9E9, 9E9, 9E9, 9E9, 9E9]];
	VAR robtarget Openhole_547 := [[434.95, -18.6, 181.12], [-0.048748, 0.705424, 0.705462, 0.048206], [0,0,0,0], [9E9, 9E9, 9E9, 9E9, 9E9, 9E9]];
	VAR robtarget Openhole_548 := [[434.46, -18.67, 181.11], [-0.050147, 0.705326, 0.70533, 0.0501], [0,0,0,0], [9E9, 9E9, 9E9, 9E9, 9E9, 9E9]];
	VAR robtarget Openhole_549 := [[433.97, -18.76, 181.1], [-0.051503, 0.705229, 0.705191, 0.052021], [0,0,0,0], [9E9, 9E9, 9E9, 9E9, 9E9, 9E9]];
	VAR robtarget Openhole_550 := [[430.5, -19.24, 181.02], [-0.061325, 0.704443, 0.704105, 0.065089], [0,0,0,0], [9E9, 9E9, 9E9, 9E9, 9E9, 9E9]];
	VAR robtarget Openhole_551 := [[429.51, -19.35, 181], [-0.064204, 0.704186, 0.70376, 0.068718], [0,0,0,0], [9E9, 9E9, 9E9, 9E9, 9E9, 9E9]];
	VAR robtarget Openhole_552 := [[429.01, -19.4, 180.99], [-0.065675, 0.70405, 0.703584, 0.070498], [0,0,0,0], [9E9, 9E9, 9E9, 9E9, 9E9, 9E9]];
	VAR robtarget Openhole_553 := [[424.02, -19.61, 180.92], [-0.081134, 0.702437, 0.7017, 0.087274], [0,0,0,0], [9E9, 9E9, 9E9, 9E9, 9E9, 9E9]];
	VAR robtarget Openhole_554 := [[422.52, -19.62, 180.91], [-0.085896, 0.70187, 0.70109, 0.092044], [0,0,0,0], [9E9, 9E9, 9E9, 9E9, 9E9, 9E9]];
	VAR robtarget Openhole_555 := [[422.02, -19.61, 180.91], [-0.08749, 0.701673, 0.700883, 0.093611], [0,0,0,0], [9E9, 9E9, 9E9, 9E9, 9E9, 9E9]];
	VAR robtarget Openhole_556 := [[407.52, -19.42, 180.9], [-0.132072, 0.694663, 0.693775, 0.13666], [0,0,0,0], [9E9, 9E9, 9E9, 9E9, 9E9, 9E9]];
	VAR robtarget Openhole_557 := [[407.02, -19.42, 180.9], [-0.133512, 0.694388, 0.693492, 0.138091], [0,0,0,0], [9E9, 9E9, 9E9, 9E9, 9E9, 9E9]];
	VAR robtarget Openhole_558 := [[398.02, -19.61, 180.77], [-0.157945, 0.689241, 0.687964, 0.16342], [0,0,0,0], [9E9, 9E9, 9E9, 9E9, 9E9, 9E9]];
	VAR robtarget Openhole_559 := [[394.34, -19.81, 180.65], [-0.167071, 0.687086, 0.685471, 0.173579], [0,0,0,0], [9E9, 9E9, 9E9, 9E9, 9E9, 9E9]];
	VAR robtarget Openhole_560 := [[362.34, -19.81, 180.69], [-0.183051, 0.683002, 0.683002, 0.183051], [0,0,0,0], [9E9, 9E9, 9E9, 9E9, 9E9, 9E9]];
	VAR robtarget Openhole_561 := [[362.35, -16.66, 182.51], [-0.183051, 0.683002, 0.683002, 0.183051], [0,0,0,0], [9E9, 9E9, 9E9, 9E9, 9E9, 9E9]];
	VAR robtarget Openhole_562 := [[389.35, -16.66, 182.43], [-0.188731, 0.681455, 0.684566, 0.177114], [0,0,0,0], [9E9, 9E9, 9E9, 9E9, 9E9, 9E9]];
	VAR robtarget Openhole_563 := [[394.35, -16.66, 182.31], [-0.176243, 0.684791, 0.687737, 0.164369], [0,0,0,0], [9E9, 9E9, 9E9, 9E9, 9E9, 9E9]];
	VAR robtarget Openhole_564 := [[395.15, -16.63, 182.31], [-0.174265, 0.685297, 0.688258, 0.162174], [0,0,0,0], [9E9, 9E9, 9E9, 9E9, 9E9, 9E9]];
	VAR robtarget Openhole_565 := [[403.65, -16.31, 182.25], [-0.152543, 0.690457, 0.693491, 0.138096], [0,0,0,0], [9E9, 9E9, 9E9, 9E9, 9E9, 9E9]];
	VAR robtarget Openhole_566 := [[410.15, -16.25, 182.11], [-0.134344, 0.694227, 0.697005, 0.119098], [0,0,0,0], [9E9, 9E9, 9E9, 9E9, 9E9, 9E9]];
	VAR robtarget Openhole_567 := [[410.65, -16.25, 182.1], [-0.132889, 0.694507, 0.697256, 0.117616], [0,0,0,0], [9E9, 9E9, 9E9, 9E9, 9E9, 9E9]];
	VAR robtarget Openhole_568 := [[425.64, -16.49, 181.64], [-0.086203, 0.701833, 0.703452, 0.071796], [0,0,0,0], [9E9, 9E9, 9E9, 9E9, 9E9, 9E9]];
	VAR robtarget Openhole_569 := [[437.63, -16.79, 181.31], [-0.045915, 0.705615, 0.70633, 0.033133], [0,0,0,0], [9E9, 9E9, 9E9, 9E9, 9E9, 9E9]];
	VAR robtarget Openhole_570 := [[438.13, -16.79, 181.3], [-0.044252, 0.705721, 0.706408, 0.031439], [0,0,0,0], [9E9, 9E9, 9E9, 9E9, 9E9, 9E9]];
	VAR robtarget Openhole_571 := [[438.63, -16.79, 181.29], [-0.042579, 0.705824, 0.706481, 0.029751], [0,0,0,0], [9E9, 9E9, 9E9, 9E9, 9E9, 9E9]];
	VAR robtarget Openhole_572 := [[440.13, -16.73, 181.27], [-0.037741, 0.706099, 0.706682, 0.024492], [0,0,0,0], [9E9, 9E9, 9E9, 9E9, 9E9, 9E9]];
	VAR robtarget Openhole_573 := [[440.62, -16.69, 181.26], [-0.036198, 0.70618, 0.706743, 0.022671], [0,0,0,0], [9E9, 9E9, 9E9, 9E9, 9E9, 9E9]];
	VAR robtarget Openhole_574 := [[441.11, -16.58, 181.26], [-0.034935, 0.706243, 0.706805, 0.020641], [0,0,0,0], [9E9, 9E9, 9E9, 9E9, 9E9, 9E9]];
	VAR robtarget Openhole_575 := [[441.66, -16.48, 181.25], [-0.033412, 0.706317, 0.706866, 0.018462], [0,0,0,0], [9E9, 9E9, 9E9, 9E9, 9E9, 9E9]];
	VAR robtarget Openhole_576 := [[443.56, -16.48, 181.2], [-0.027008, 0.706591, 0.707005, 0.012019], [0,0,0,0], [9E9, 9E9, 9E9, 9E9, 9E9, 9E9]];
	VAR robtarget Openhole_577 := [[443.93, -15.46, 181.25], [-0.029222, 0.706503, 0.70707, 0.007254], [0,0,0,0], [9E9, 9E9, 9E9, 9E9, 9E9, 9E9]];
	VAR robtarget Openhole_578 := [[442.03, -15.46, 181.31], [-0.035624, 0.706209, 0.706974, 0.013704], [0,0,0,0], [9E9, 9E9, 9E9, 9E9, 9E9, 9E9]];
	VAR robtarget Openhole_579 := [[441.46, -15.51, 181.33], [-0.037375, 0.706118, 0.70693, 0.015821], [0,0,0,0], [9E9, 9E9, 9E9, 9E9, 9E9, 9E9]];
	VAR robtarget Openhole_580 := [[440.97, -15.59, 181.34], [-0.038741, 0.706045, 0.706883, 0.017785], [0,0,0,0], [9E9, 9E9, 9E9, 9E9, 9E9, 9E9]];
	VAR robtarget Openhole_581 := [[439.97, -15.62, 181.37], [-0.042, 0.705858, 0.706787, 0.021272], [0,0,0,0], [9E9, 9E9, 9E9, 9E9, 9E9, 9E9]];
	VAR robtarget Openhole_582 := [[439.47, -15.62, 181.39], [-0.043689, 0.705756, 0.706734, 0.022951], [0,0,0,0], [9E9, 9E9, 9E9, 9E9, 9E9, 9E9]];
	VAR robtarget Openhole_583 := [[438.97, -15.61, 181.4], [-0.045413, 0.705647, 0.706679, 0.024591], [0,0,0,0], [9E9, 9E9, 9E9, 9E9, 9E9, 9E9]];
	VAR robtarget Openhole_584 := [[438.47, -15.58, 181.42], [-0.047169, 0.705532, 0.706622, 0.026192], [0,0,0,0], [9E9, 9E9, 9E9, 9E9, 9E9, 9E9]];
	VAR robtarget Openhole_585 := [[437.48, -15.49, 181.47], [-0.050785, 0.705281, 0.706501, 0.029259], [0,0,0,0], [9E9, 9E9, 9E9, 9E9, 9E9, 9E9]];
	VAR robtarget Openhole_586 := [[431.51, -14.94, 181.76], [-0.07236, 0.703395, 0.705519, 0.047357], [0,0,0,0], [9E9, 9E9, 9E9, 9E9, 9E9, 9E9]];
	VAR robtarget Openhole_587 := [[422.53, -14.66, 182.19], [-0.102032, 0.699707, 0.703034, 0.075783], [0,0,0,0], [9E9, 9E9, 9E9, 9E9, 9E9, 9E9]];
	VAR robtarget Openhole_588 := [[413.53, -14.6, 182.59], [-0.129596, 0.695129, 0.699461, 0.103706], [0,0,0,0], [9E9, 9E9, 9E9, 9E9, 9E9, 9E9]];
	VAR robtarget Openhole_589 := [[413.04, -14.6, 182.61], [-0.131067, 0.694854, 0.699233, 0.105227], [0,0,0,0], [9E9, 9E9, 9E9, 9E9, 9E9, 9E9]];
	VAR robtarget Openhole_590 := [[401.54, -14.77, 183.02], [-0.162952, 0.688075, 0.69325, 0.139302], [0,0,0,0], [9E9, 9E9, 9E9, 9E9, 9E9, 9E9]];
	VAR robtarget Openhole_591 := [[394.35, -15.07, 183.15], [-0.180853, 0.683588, 0.688833, 0.159717], [0,0,0,0], [9E9, 9E9, 9E9, 9E9, 9E9, 9E9]];
	VAR robtarget Openhole_592 := [[389.35, -15.07, 183.34], [-0.193225, 0.680194, 0.685724, 0.172577], [0,0,0,0], [9E9, 9E9, 9E9, 9E9, 9E9, 9E9]];
	VAR robtarget Openhole_593 := [[362.35, -15.07, 183.43], [-0.183051, 0.683002, 0.683002, 0.183051], [0,0,0,0], [9E9, 9E9, 9E9, 9E9, 9E9, 9E9]];
	VAR robtarget Openhole_594 := [[362.35, -14.11, 183.99], [-0.183051, 0.683002, 0.683002, 0.183051], [0,0,0,0], [9E9, 9E9, 9E9, 9E9, 9E9, 9E9]];
	VAR robtarget Openhole_595 := [[389.35, -14.11, 183.9], [-0.195953, 0.679413, 0.686413, 0.169816], [0,0,0,0], [9E9, 9E9, 9E9, 9E9, 9E9, 9E9]];
	VAR robtarget Openhole_596 := [[394.35, -14.11, 183.66], [-0.18365, 0.682842, 0.689483, 0.156887], [0,0,0,0], [9E9, 9E9, 9E9, 9E9, 9E9, 9E9]];
	VAR robtarget Openhole_597 := [[404.57, -13.71, 183.35], [-0.157908, 0.68925, 0.695516, 0.127507], [0,0,0,0], [9E9, 9E9, 9E9, 9E9, 9E9, 9E9]];
	VAR robtarget Openhole_598 := [[419.55, -13.55, 182.63], [-0.114842, 0.697719, 0.702379, 0.081629], [0,0,0,0], [9E9, 9E9, 9E9, 9E9, 9E9, 9E9]];
	VAR robtarget Openhole_599 := [[420.05, -13.55, 182.61], [-0.11331, 0.697969, 0.702561, 0.080046], [0,0,0,0], [9E9, 9E9, 9E9, 9E9, 9E9, 9E9]];
	VAR robtarget Openhole_600 := [[430.53, -13.69, 182.03], [-0.079678, 0.702603, 0.70558, 0.046444], [0,0,0,0], [9E9, 9E9, 9E9, 9E9, 9E9, 9E9]];
	VAR robtarget Openhole_601 := [[435.51, -14.05, 181.72], [-0.062177, 0.704368, 0.706427, 0.030998], [0,0,0,0], [9E9, 9E9, 9E9, 9E9, 9E9, 9E9]];
	VAR robtarget Openhole_602 := [[438.48, -14.4, 181.54], [-0.051087, 0.705259, 0.706759, 0.022176], [0,0,0,0], [9E9, 9E9, 9E9, 9E9, 9E9, 9E9]];
	VAR robtarget Openhole_603 := [[438.98, -14.45, 181.52], [-0.04928, 0.705387, 0.706806, 0.020638], [0,0,0,0], [9E9, 9E9, 9E9, 9E9, 9E9, 9E9]];
	VAR robtarget Openhole_604 := [[439.48, -14.47, 181.49], [-0.047521, 0.705508, 0.70685, 0.019038], [0,0,0,0], [9E9, 9E9, 9E9, 9E9, 9E9, 9E9]];
	VAR robtarget Openhole_605 := [[439.98, -14.49, 181.47], [-0.045811, 0.705621, 0.706893, 0.017382], [0,0,0,0], [9E9, 9E9, 9E9, 9E9, 9E9, 9E9]];
	VAR robtarget Openhole_606 := [[440.98, -14.49, 181.43], [-0.042441, 0.705832, 0.706968, 0.014009], [0,0,0,0], [9E9, 9E9, 9E9, 9E9, 9E9, 9E9]];
	VAR robtarget Openhole_607 := [[441.98, -14.53, 181.38], [-0.038942, 0.706034, 0.707025, 0.010759], [0,0,0,0], [9E9, 9E9, 9E9, 9E9, 9E9, 9E9]];
	VAR robtarget Openhole_608 := [[442.51, -14.54, 181.36], [-0.037101, 0.706133, 0.70705, 0.008985], [0,0,0,0], [9E9, 9E9, 9E9, 9E9, 9E9, 9E9]];
	VAR robtarget Openhole_609 := [[444.28, -14.54, 181.28], [-0.031112, 0.706422, 0.707101, 0.002945], [0,0,0,0], [9E9, 9E9, 9E9, 9E9, 9E9, 9E9]];
	VAR robtarget Openhole_610 := [[445.21, -13.31, 181.29], [-0.032163, 0.706375, 0.707093, -0.0044], [0,0,0,0], [9E9, 9E9, 9E9, 9E9, 9E9, 9E9]];
	VAR robtarget Openhole_611 := [[443.43, -13.31, 181.39], [-0.038155, 0.706077, 0.707105, 0.001648], [0,0,0,0], [9E9, 9E9, 9E9, 9E9, 9E9, 9E9]];
	VAR robtarget Openhole_612 := [[442.74, -13.1, 181.44], [-0.041181, 0.705907, 0.707099, 0.003297], [0,0,0,0], [9E9, 9E9, 9E9, 9E9, 9E9, 9E9]];
	VAR robtarget Openhole_613 := [[440.25, -13.05, 181.59], [-0.049758, 0.705354, 0.707012, 0.011589], [0,0,0,0], [9E9, 9E9, 9E9, 9E9, 9E9, 9E9]];
	VAR robtarget Openhole_614 := [[433.78, -12.57, 182.03], [-0.072797, 0.70335, 0.706389, 0.03185], [0,0,0,0], [9E9, 9E9, 9E9, 9E9, 9E9, 9E9]];
	VAR robtarget Openhole_615 := [[427.8, -12.45, 182.42], [-0.092579, 0.70102, 0.705238, 0.051376], [0,0,0,0], [9E9, 9E9, 9E9, 9E9, 9E9, 9E9]];
	VAR robtarget Openhole_616 := [[427.3, -12.45, 182.46], [-0.094171, 0.700808, 0.705116, 0.053019], [0,0,0,0], [9E9, 9E9, 9E9, 9E9, 9E9, 9E9]];
	VAR robtarget Openhole_617 := [[408.83, -12.69, 183.53], [-0.149167, 0.691194, 0.698203, 0.111858], [0,0,0,0], [9E9, 9E9, 9E9, 9E9, 9E9, 9E9]];
	VAR robtarget Openhole_618 := [[397.35, -13.06, 184.05], [-0.179073, 0.684056, 0.69192, 0.145761], [0,0,0,0], [9E9, 9E9, 9E9, 9E9, 9E9, 9E9]];
	VAR robtarget Openhole_619 := [[394.33, -13.23, 184.13], [-0.186259, 0.682135, 0.690055, 0.154352], [0,0,0,0], [9E9, 9E9, 9E9, 9E9, 9E9, 9E9]];
	VAR robtarget Openhole_620 := [[389.36, -13.23, 184.41], [-0.198445, 0.67869, 0.687033, 0.167288], [0,0,0,0], [9E9, 9E9, 9E9, 9E9, 9E9, 9E9]];
	VAR robtarget Openhole_621 := [[362.36, -13.23, 184.5], [-0.183051, 0.683002, 0.683002, 0.183051], [0,0,0,0], [9E9, 9E9, 9E9, 9E9, 9E9, 9E9]];
	VAR robtarget Openhole_622 := [[362.36, -12.34, 185.01], [-0.183051, 0.683002, 0.683002, 0.183051], [0,0,0,0], [9E9, 9E9, 9E9, 9E9, 9E9, 9E9]];
	VAR robtarget Openhole_623 := [[374.36, -12.34, 184.97], [-0.183051, 0.683002, 0.683002, 0.183051], [0,0,0,0], [9E9, 9E9, 9E9, 9E9, 9E9, 9E9]];
	VAR robtarget Openhole_624 := [[389.36, -12.34, 184.92], [-0.200934, 0.677957, 0.687644, 0.164758], [0,0,0,0], [9E9, 9E9, 9E9, 9E9, 9E9, 9E9]];
	VAR robtarget Openhole_625 := [[394.34, -12.34, 184.6], [-0.188806, 0.681434, 0.690631, 0.151754], [0,0,0,0], [9E9, 9E9, 9E9, 9E9, 9E9, 9E9]];
	VAR robtarget Openhole_626 := [[404.83, -11.88, 184.12], [-0.162742, 0.688124, 0.696657, 0.121118], [0,0,0,0], [9E9, 9E9, 9E9, 9E9, 9E9, 9E9]];
	VAR robtarget Openhole_627 := [[429.78, -11.27, 182.52], [-0.090141, 0.701338, 0.705924, 0.040884], [0,0,0,0], [9E9, 9E9, 9E9, 9E9, 9E9, 9E9]];
	VAR robtarget Openhole_628 := [[431.77, -11.25, 182.38], [-0.083747, 0.70213, 0.70628, 0.034177], [0,0,0,0], [9E9, 9E9, 9E9, 9E9, 9E9, 9E9]];
	VAR robtarget Openhole_629 := [[432.27, -11.25, 182.34], [-0.082125, 0.702321, 0.706359, 0.032508], [0,0,0,0], [9E9, 9E9, 9E9, 9E9, 9E9, 9E9]];
	VAR robtarget Openhole_630 := [[441.74, -11.43, 181.62], [-0.050214, 0.705322, 0.707106, 0.001035], [0,0,0,0], [9E9, 9E9, 9E9, 9E9, 9E9, 9E9]];
	VAR robtarget Openhole_631 := [[442.24, -11.45, 181.58], [-0.048453, 0.705445, 0.707107, -0.000573], [0,0,0,0], [9E9, 9E9, 9E9, 9E9, 9E9, 9E9]];
	VAR robtarget Openhole_632 := [[443.23, -11.52, 181.5], [-0.044865, 0.705682, 0.707097, -0.003718], [0,0,0,0], [9E9, 9E9, 9E9, 9E9, 9E9, 9E9]];
	VAR robtarget Openhole_633 := [[444.22, -11.62, 181.43], [-0.041189, 0.705906, 0.707074, -0.006769], [0,0,0,0], [9E9, 9E9, 9E9, 9E9, 9E9, 9E9]];
	VAR robtarget Openhole_634 := [[444.72, -11.69, 181.39], [-0.039307, 0.706013, 0.707059, -0.008244], [0,0,0,0], [9E9, 9E9, 9E9, 9E9, 9E9, 9E9]];
	VAR robtarget Openhole_635 := [[445.25, -11.83, 181.35], [-0.037027, 0.706137, 0.707042, -0.009588], [0,0,0,0], [9E9, 9E9, 9E9, 9E9, 9E9, 9E9]];
	VAR robtarget Openhole_636 := [[454.82, -12.87, 180.74], [-0.001006, 0.707106, 0.706051, -0.038624], [0,0,0,0], [9E9, 9E9, 9E9, 9E9, 9E9, 9E9]];
	VAR robtarget Openhole_637 := [[455.35, -12.53, 180.69], [-0.000351, 0.707107, 0.705884, -0.041572], [0,0,0,0], [9E9, 9E9, 9E9, 9E9, 9E9, 9E9]];
	VAR robtarget Openhole_638 := [[455.8, -12.3, 180.64], [0.000386, 0.707107, 0.705746, -0.043839], [0,0,0,0], [9E9, 9E9, 9E9, 9E9, 9E9, 9E9]];
	VAR robtarget Openhole_639 := [[456.25, -12.09, 180.6], [0.001198, 0.707106, 0.705604, -0.04608], [0,0,0,0], [9E9, 9E9, 9E9, 9E9, 9E9, 9E9]];
	VAR robtarget Openhole_640 := [[456.7, -11.89, 180.56], [0.002048, 0.707104, 0.705455, -0.048302], [0,0,0,0], [9E9, 9E9, 9E9, 9E9, 9E9, 9E9]];
	VAR robtarget Openhole_641 := [[457.17, -11.7, 180.51], [0.003007, 0.7071, 0.705303, -0.050478], [0,0,0,0], [9E9, 9E9, 9E9, 9E9, 9E9, 9E9]];
	VAR robtarget Openhole_642 := [[458.11, -11.38, 180.42], [0.005095, 0.707088, 0.704985, -0.054742], [0,0,0,0], [9E9, 9E9, 9E9, 9E9, 9E9, 9E9]];
	VAR robtarget Openhole_643 := [[464.29, -9.52, 179.69], [0.019804, 0.706829, 0.702395, -0.081491], [0,0,0,0], [9E9, 9E9, 9E9, 9E9, 9E9, 9E9]];
	VAR robtarget Openhole_644 := [[464.77, -9.39, 179.63], [0.020974, 0.706796, 0.70216, -0.083496], [0,0,0,0], [9E9, 9E9, 9E9, 9E9, 9E9, 9E9]];
	VAR robtarget Openhole_645 := [[469.6, -8.3, 178.97], [0.033532, 0.706311, 0.699606, -0.10272], [0,0,0,0], [9E9, 9E9, 9E9, 9E9, 9E9, 9E9]];
	VAR robtarget Openhole_646 := [[474.02, -7.68, 178.37], [0.046079, 0.705604, 0.69708, -0.118657], [0,0,0,0], [9E9, 9E9, 9E9, 9E9, 9E9, 9E9]];
	VAR robtarget Openhole_647 := [[478.47, -7.38, 177.8], [0.059627, 0.704588, 0.694441, -0.133235], [0,0,0,0], [9E9, 9E9, 9E9, 9E9, 9E9, 9E9]];
	VAR robtarget Openhole_648 := [[480.96, -7.35, 177.51], [0.067492, 0.703878, 0.692955, -0.140759], [0,0,0,0], [9E9, 9E9, 9E9, 9E9, 9E9, 9E9]];
	VAR robtarget Openhole_649 := [[481.45, -7.35, 177.45], [0.069079, 0.703724, 0.692656, -0.142226], [0,0,0,0], [9E9, 9E9, 9E9, 9E9, 9E9, 9E9]];
	VAR robtarget Openhole_650 := [[487.92, -7.59, 176.82], [0.09003, 0.701352, 0.688739, -0.160122], [0,0,0,0], [9E9, 9E9, 9E9, 9E9, 9E9, 9E9]];
	VAR robtarget Openhole_651 := [[499.85, -8.3, 175.85], [0.127355, 0.695544, 0.681113, -0.189959], [0,0,0,0], [9E9, 9E9, 9E9, 9E9, 9E9, 9E9]];
	VAR robtarget Openhole_652 := [[501.35, -8.33, 175.7], [0.131609, 0.694751, 0.680072, -0.193655], [0,0,0,0], [9E9, 9E9, 9E9, 9E9, 9E9, 9E9]];
	VAR robtarget Openhole_653 := [[501.85, -8.33, 175.65], [0.13299, 0.694488, 0.679716, -0.1949], [0,0,0,0], [9E9, 9E9, 9E9, 9E9, 9E9, 9E9]];
	VAR robtarget Openhole_654 := [[503.83, -8.3, 175.44], [0.13839, 0.693432, 0.678268, -0.199882], [0,0,0,0], [9E9, 9E9, 9E9, 9E9, 9E9, 9E9]];
	VAR robtarget Openhole_655 := [[504.35, -8.28, 175.37], [0.139727, 0.693164, 0.677869, -0.201229], [0,0,0,0], [9E9, 9E9, 9E9, 9E9, 9E9, 9E9]];
	VAR robtarget Openhole_656 := [[509.33, -8.28, 174.85], [0.183051, 0.683002, 0.683002, -0.183051], [0,0,0,0], [9E9, 9E9, 9E9, 9E9, 9E9, 9E9]];
	VAR robtarget Openhole_657 := [[536.33, -8.27, 174.77], [0.183051, 0.683002, 0.683002, -0.183051], [0,0,0,0], [9E9, 9E9, 9E9, 9E9, 9E9, 9E9]];
	VAR robtarget Openhole_658 := [[536.33, -9.15, 175.27], [0.183051, 0.683002, 0.683002, -0.183051], [0,0,0,0], [9E9, 9E9, 9E9, 9E9, 9E9, 9E9]];
	VAR robtarget Openhole_659 := [[509.33, -9.15, 175.36], [0.183051, 0.683002, 0.683002, -0.183051], [0,0,0,0], [9E9, 9E9, 9E9, 9E9, 9E9, 9E9]];
	VAR robtarget Openhole_660 := [[504.33, -9.15, 175.83], [0.142198, 0.692661, 0.678622, -0.198677], [0,0,0,0], [9E9, 9E9, 9E9, 9E9, 9E9, 9E9]];
	VAR robtarget Openhole_661 := [[503.69, -9.17, 175.91], [0.140537, 0.693, 0.679103, -0.197026], [0,0,0,0], [9E9, 9E9, 9E9, 9E9, 9E9, 9E9]];
	VAR robtarget Openhole_662 := [[503.19, -9.2, 175.97], [0.139282, 0.693254, 0.679483, -0.195711], [0,0,0,0], [9E9, 9E9, 9E9, 9E9, 9E9, 9E9]];
	VAR robtarget Openhole_663 := [[500.21, -9.26, 176.28], [0.131202, 0.694828, 0.681641, -0.188057], [0,0,0,0], [9E9, 9E9, 9E9, 9E9, 9E9, 9E9]];
	VAR robtarget Openhole_664 := [[499.71, -9.26, 176.32], [0.1298, 0.695091, 0.681989, -0.186793], [0,0,0,0], [9E9, 9E9, 9E9, 9E9, 9E9, 9E9]];
	VAR robtarget Openhole_665 := [[491.74, -8.94, 176.94], [0.105788, 0.699149, 0.687196, -0.166617], [0,0,0,0], [9E9, 9E9, 9E9, 9E9, 9E9, 9E9]];
	VAR robtarget Openhole_666 := [[482.78, -8.57, 177.69], [0.077159, 0.702884, 0.692637, -0.142317], [0,0,0,0], [9E9, 9E9, 9E9, 9E9, 9E9, 9E9]];
	VAR robtarget Openhole_667 := [[481.79, -8.56, 177.79], [0.073999, 0.703224, 0.693229, -0.139402], [0,0,0,0], [9E9, 9E9, 9E9, 9E9, 9E9, 9E9]];
	VAR robtarget Openhole_668 := [[481.29, -8.56, 177.84], [0.072428, 0.703388, 0.693525, -0.137924], [0,0,0,0], [9E9, 9E9, 9E9, 9E9, 9E9, 9E9]];
	VAR robtarget Openhole_669 := [[476.32, -8.73, 178.39], [0.057031, 0.704803, 0.696437, -0.122377], [0,0,0,0], [9E9, 9E9, 9E9, 9E9, 9E9, 9E9]];
	VAR robtarget Openhole_670 := [[471.89, -9.23, 178.94], [0.044155, 0.705727, 0.698977, -0.10692], [0,0,0,0], [9E9, 9E9, 9E9, 9E9, 9E9, 9E9]];
	VAR robtarget Openhole_671 := [[468.97, -9.8, 179.32], [0.036353, 0.706172, 0.700593, -0.095755], [0,0,0,0], [9E9, 9E9, 9E9, 9E9, 9E9, 9E9]];
	VAR robtarget Openhole_672 := [[466.57, -10.43, 179.64], [0.030434, 0.706452, 0.701867, -0.085926], [0,0,0,0], [9E9, 9E9, 9E9, 9E9, 9E9, 9E9]];
	VAR robtarget Openhole_673 := [[463.74, -11.36, 180], [0.024094, 0.706696, 0.703272, -0.073543], [0,0,0,0], [9E9, 9E9, 9E9, 9E9, 9E9, 9E9]];
	VAR robtarget Openhole_674 := [[461.9, -12.1, 180.22], [0.020361, 0.706814, 0.704116, -0.064963], [0,0,0,0], [9E9, 9E9, 9E9, 9E9, 9E9, 9E9]];
	VAR robtarget Openhole_675 := [[460.53, -12.71, 180.38], [0.017798, 0.706883, 0.704692, -0.058384], [0,0,0,0], [9E9, 9E9, 9E9, 9E9, 9E9, 9E9]];
	VAR robtarget Openhole_676 := [[459.64, -13.14, 180.48], [0.016238, 0.70692, 0.705048, -0.053924], [0,0,0,0], [9E9, 9E9, 9E9, 9E9, 9E9, 9E9]];
	VAR robtarget Openhole_677 := [[459.2, -13.37, 180.53], [0.015518, 0.706936, 0.705217, -0.051669], [0,0,0,0], [9E9, 9E9, 9E9, 9E9, 9E9, 9E9]];
	VAR robtarget Openhole_678 := [[458.76, -13.61, 180.57], [0.014842, 0.706951, 0.705379, -0.049396], [0,0,0,0], [9E9, 9E9, 9E9, 9E9, 9E9, 9E9]];
	VAR robtarget Openhole_679 := [[457.91, -14.13, 180.66], [0.01369, 0.706974, 0.705687, -0.044787], [0,0,0,0], [9E9, 9E9, 9E9, 9E9, 9E9, 9E9]];
	VAR robtarget Openhole_680 := [[456.45, -15.03, 180.79], [0.011828, 0.707008, 0.706148, -0.036814], [0,0,0,0], [9E9, 9E9, 9E9, 9E9, 9E9, 9E9]];
	VAR robtarget Openhole_681 := [[454.01, -15.03, 180.88], [0.003529, 0.707098, 0.706531, -0.028522], [0,0,0,0], [9E9, 9E9, 9E9, 9E9, 9E9, 9E9]];
	VAR robtarget Openhole_682 := [[454.58, -16.45, 180.93], [0.010279, 0.707032, 0.706642, -0.025621], [0,0,0,0], [9E9, 9E9, 9E9, 9E9, 9E9, 9E9]];
	VAR robtarget Openhole_683 := [[457.02, -16.45, 180.87], [0.018565, 0.706863, 0.706293, -0.033915], [0,0,0,0], [9E9, 9E9, 9E9, 9E9, 9E9, 9E9]];
	VAR robtarget Openhole_684 := [[457.6, -16.2, 180.84], [0.019651, 0.706834, 0.706153, -0.036721], [0,0,0,0], [9E9, 9E9, 9E9, 9E9, 9E9, 9E9]];
	VAR robtarget Openhole_685 := [[458.48, -15.74, 180.77], [0.02109, 0.706792, 0.705902, -0.041268], [0,0,0,0], [9E9, 9E9, 9E9, 9E9, 9E9, 9E9]];
	VAR robtarget Openhole_686 := [[458.92, -15.49, 180.74], [0.021714, 0.706773, 0.705763, -0.043565], [0,0,0,0], [9E9, 9E9, 9E9, 9E9, 9E9, 9E9]];
	VAR robtarget Openhole_687 := [[459.34, -15.23, 180.7], [0.022265, 0.706756, 0.705617, -0.045876], [0,0,0,0], [9E9, 9E9, 9E9, 9E9, 9E9, 9E9]];
	VAR robtarget Openhole_688 := [[460.18, -14.69, 180.61], [0.023265, 0.706724, 0.7053, -0.050512], [0,0,0,0], [9E9, 9E9, 9E9, 9E9, 9E9, 9E9]];
	VAR robtarget Openhole_689 := [[461.03, -14.18, 180.52], [0.024437, 0.706684, 0.704957, -0.055093], [0,0,0,0], [9E9, 9E9, 9E9, 9E9, 9E9, 9E9]];
	VAR robtarget Openhole_690 := [[463.23, -13.02, 180.26], [0.02793, 0.706555, 0.70399, -0.066314], [0,0,0,0], [9E9, 9E9, 9E9, 9E9, 9E9, 9E9]];
	VAR robtarget Openhole_691 := [[463.68, -12.81, 180.2], [0.028731, 0.706523, 0.70378, -0.068511], [0,0,0,0], [9E9, 9E9, 9E9, 9E9, 9E9, 9E9]];
	VAR robtarget Openhole_692 := [[465.05, -12.22, 180.03], [0.031347, 0.706412, 0.703119, -0.074993], [0,0,0,0], [9E9, 9E9, 9E9, 9E9, 9E9, 9E9]];
	VAR robtarget Openhole_693 := [[465.51, -12.04, 179.97], [0.032289, 0.706369, 0.702889, -0.077114], [0,0,0,0], [9E9, 9E9, 9E9, 9E9, 9E9, 9E9]];
